// ---- DUTs/IO/PdoEntries/Control_FF5AB9B2.TcDUT
{attribute 'GeneratedUsingTerminal: EJ7334-0008-0016'}
{attribute addProperty BoxType "EJ7334-0008-0016"}
{attribute addProperty Id "EnableBOOL1ResetBOOL1"}
{attribute addProperty CRC "4284135858"}
{attribute addProperty Size "2"}
TYPE Control_FF5AB9B2 :
STRUCT
	{attribute addProperty Name "Enable"}
	Enable : BOOL;
	{attribute addProperty Name "Reset"}
	Reset : BOOL;
END_STRUCT
END_TYPE

// ---- DUTs/IO/PdoEntries/FSOE_1F44E1B4.TcDUT
{attribute 'GeneratedUsingTerminal: EJ1914-0000-0017'}
{attribute addProperty BoxType "EJ1914-0000-0017"}
{attribute addProperty Id "FSoE_CommandUSINT1FSIN_Module_1_Channel_1_InputBOOL1FSIN_Module_1_Channel_2_InputBOOL1FSIN_Module_1_Module_FaultBOOL1FSIN_Module_2_Channel_1_InputBOOL1FSIN_Module_2_Channel_2_InputBOOL1FSIN_Module_2_Module_FaultBOOL1FSoE_CRC_000UINT2FSoE_Connection_IDUINT2"}
{attribute addProperty CRC "524607924"}
{attribute addProperty Size "11"}
TYPE FSOE_1F44E1B4 :
STRUCT
	{attribute addProperty Name "FSoE_Command"}
	FSoE_Command : USINT;
	{attribute addProperty Name "FSIN_Module_1_Channel_1_Input"}
	FSIN_Module_1_Channel_1_Input : BOOL;
	{attribute addProperty Name "FSIN_Module_1_Channel_2_Input"}
	FSIN_Module_1_Channel_2_Input : BOOL;
	{attribute addProperty Name "FSIN_Module_1_Module_Fault"}
	FSIN_Module_1_Module_Fault : BOOL;
	{attribute addProperty Name "FSIN_Module_2_Channel_1_Input"}
	FSIN_Module_2_Channel_1_Input : BOOL;
	{attribute addProperty Name "FSIN_Module_2_Channel_2_Input"}
	FSIN_Module_2_Channel_2_Input : BOOL;
	{attribute addProperty Name "FSIN_Module_2_Module_Fault"}
	FSIN_Module_2_Module_Fault : BOOL;
	{attribute addProperty Name "FSoE_CRC_000"}
	FSoE_CRC_000 : UINT;
	{attribute addProperty Name "FSoE_Connection_ID"}
	FSoE_Connection_ID : UINT;
END_STRUCT
END_TYPE

// ---- DUTs/IO/PdoEntries/FSOE_9A7ED3DD.TcDUT
{attribute 'GeneratedUsingTerminal: EJ1914-0000-0017'}
{attribute addProperty BoxType "EJ1914-0000-0017"}
{attribute addProperty Id "FSoE_CommandUSINT1FSIN_Module_1_ErrAckBOOL1FSIN_Module_2_ErrAckBOOL1FSoE_CRC_000UINT2FSoE_Connection_IDUINT2"}
{attribute addProperty CRC "2592003037"}
{attribute addProperty Size "7"}
TYPE FSOE_9A7ED3DD :
STRUCT
	{attribute addProperty Name "FSoE_Command"}
	FSoE_Command : USINT;
	{attribute addProperty Name "FSIN_Module_1_ErrAck"}
	FSIN_Module_1_ErrAck : BOOL;
	{attribute addProperty Name "FSIN_Module_2_ErrAck"}
	FSIN_Module_2_ErrAck : BOOL;
	{attribute addProperty Name "FSoE_CRC_000"}
	FSoE_CRC_000 : UINT;
	{attribute addProperty Name "FSoE_Connection_ID"}
	FSoE_Connection_ID : UINT;
END_STRUCT
END_TYPE

// ---- DUTs/IO/PdoEntries/FSOE_9F04885D.TcDUT
{attribute 'GeneratedUsingTerminal: EJ1918-0000-0017'}
{attribute addProperty BoxType "EJ1918-0000-0017"}
{attribute addProperty Id "FSoE_CommandUSINT1FSIN_Module_1_Channel_1_InputBOOL1FSIN_Module_1_Channel_2_InputBOOL1FSIN_Module_1_Module_FaultBOOL1FSIN_Module_2_Channel_1_InputBOOL1FSIN_Module_2_Channel_2_InputBOOL1FSIN_Module_2_Module_FaultBOOL1FSIN_Module_3_Channel_1_InputBOOL1FSIN_Module_3_Channel_2_InputBOOL1FSIN_Module_3_Module_FaultBOOL1FSIN_Module_4_Channel_1_InputBOOL1FSIN_Module_4_Channel_2_InputBOOL1FSIN_Module_4_Module_FaultBOOL1FSoE_CRC_000UINT2FSoE_Connection_IDUINT2"}
{attribute addProperty CRC "2667874397"}
{attribute addProperty Size "17"}
TYPE FSOE_9F04885D :
STRUCT
	{attribute addProperty Name "FSoE_Command"}
	FSoE_Command : USINT;
	{attribute addProperty Name "FSIN_Module_1_Channel_1_Input"}
	FSIN_Module_1_Channel_1_Input : BOOL;
	{attribute addProperty Name "FSIN_Module_1_Channel_2_Input"}
	FSIN_Module_1_Channel_2_Input : BOOL;
	{attribute addProperty Name "FSIN_Module_1_Module_Fault"}
	FSIN_Module_1_Module_Fault : BOOL;
	{attribute addProperty Name "FSIN_Module_2_Channel_1_Input"}
	FSIN_Module_2_Channel_1_Input : BOOL;
	{attribute addProperty Name "FSIN_Module_2_Channel_2_Input"}
	FSIN_Module_2_Channel_2_Input : BOOL;
	{attribute addProperty Name "FSIN_Module_2_Module_Fault"}
	FSIN_Module_2_Module_Fault : BOOL;
	{attribute addProperty Name "FSIN_Module_3_Channel_1_Input"}
	FSIN_Module_3_Channel_1_Input : BOOL;
	{attribute addProperty Name "FSIN_Module_3_Channel_2_Input"}
	FSIN_Module_3_Channel_2_Input : BOOL;
	{attribute addProperty Name "FSIN_Module_3_Module_Fault"}
	FSIN_Module_3_Module_Fault : BOOL;
	{attribute addProperty Name "FSIN_Module_4_Channel_1_Input"}
	FSIN_Module_4_Channel_1_Input : BOOL;
	{attribute addProperty Name "FSIN_Module_4_Channel_2_Input"}
	FSIN_Module_4_Channel_2_Input : BOOL;
	{attribute addProperty Name "FSIN_Module_4_Module_Fault"}
	FSIN_Module_4_Module_Fault : BOOL;
	{attribute addProperty Name "FSoE_CRC_000"}
	FSoE_CRC_000 : UINT;
	{attribute addProperty Name "FSoE_Connection_ID"}
	FSoE_Connection_ID : UINT;
END_STRUCT
END_TYPE

// ---- DUTs/IO/PdoEntries/FSOE_87848461.TcDUT
{attribute 'GeneratedUsingTerminal: EJ1918-0000-0017'}
{attribute addProperty BoxType "EJ1918-0000-0017"}
{attribute addProperty Id "FSoE_CommandUSINT1FSIN_Module_1_ErrAckBOOL1FSIN_Module_2_ErrAckBOOL1FSIN_Module_3_ErrAckBOOL1FSIN_Module_4_ErrAckBOOL1FSoE_CRC_000UINT2FSoE_Connection_IDUINT2"}
{attribute addProperty CRC "2273608801"}
{attribute addProperty Size "9"}
TYPE FSOE_87848461 :
STRUCT
	{attribute addProperty Name "FSoE_Command"}
	FSoE_Command : USINT;
	{attribute addProperty Name "FSIN_Module_1_ErrAck"}
	FSIN_Module_1_ErrAck : BOOL;
	{attribute addProperty Name "FSIN_Module_2_ErrAck"}
	FSIN_Module_2_ErrAck : BOOL;
	{attribute addProperty Name "FSIN_Module_3_ErrAck"}
	FSIN_Module_3_ErrAck : BOOL;
	{attribute addProperty Name "FSIN_Module_4_ErrAck"}
	FSIN_Module_4_ErrAck : BOOL;
	{attribute addProperty Name "FSoE_CRC_000"}
	FSoE_CRC_000 : UINT;
	{attribute addProperty Name "FSoE_Connection_ID"}
	FSoE_Connection_ID : UINT;
END_STRUCT
END_TYPE

// ---- DUTs/IO/PdoEntries/FSOE_BBC930F7.TcDUT
{attribute 'GeneratedUsingTerminal: EJ1957-0000-0017'}
{attribute addProperty BoxType "EJ1957-0000-0017"}
{attribute addProperty Id "FSoE_CommandUSINT1FSOUT_Module_Module_FaultBOOL1FSIN_Module_1_Channel_1_InputBOOL1FSIN_Module_1_Channel_2_InputBOOL1FSIN_Module_1_Module_FaultBOOL1FSIN_Module_2_Channel_1_InputBOOL1FSIN_Module_2_Channel_2_InputBOOL1FSIN_Module_2_Module_FaultBOOL1FSIN_Module_3_Channel_1_InputBOOL1FSIN_Module_3_Channel_2_InputBOOL1FSIN_Module_3_Module_FaultBOOL1FSIN_Module_4_Channel_1_InputBOOL1FSIN_Module_4_Channel_2_InputBOOL1FSIN_Module_4_Module_FaultBOOL1FSoE_CRC_000UINT2FSoE_Connection_IDUINT2"}
{attribute addProperty CRC "3150524663"}
{attribute addProperty Size "18"}
TYPE FSOE_BBC930F7 :
STRUCT
	{attribute addProperty Name "FSoE_Command"}
	FSoE_Command : USINT;
	{attribute addProperty Name "FSOUT_Module_Module_Fault"}
	FSOUT_Module_Module_Fault : BOOL;
	{attribute addProperty Name "FSIN_Module_1_Channel_1_Input"}
	FSIN_Module_1_Channel_1_Input : BOOL;
	{attribute addProperty Name "FSIN_Module_1_Channel_2_Input"}
	FSIN_Module_1_Channel_2_Input : BOOL;
	{attribute addProperty Name "FSIN_Module_1_Module_Fault"}
	FSIN_Module_1_Module_Fault : BOOL;
	{attribute addProperty Name "FSIN_Module_2_Channel_1_Input"}
	FSIN_Module_2_Channel_1_Input : BOOL;
	{attribute addProperty Name "FSIN_Module_2_Channel_2_Input"}
	FSIN_Module_2_Channel_2_Input : BOOL;
	{attribute addProperty Name "FSIN_Module_2_Module_Fault"}
	FSIN_Module_2_Module_Fault : BOOL;
	{attribute addProperty Name "FSIN_Module_3_Channel_1_Input"}
	FSIN_Module_3_Channel_1_Input : BOOL;
	{attribute addProperty Name "FSIN_Module_3_Channel_2_Input"}
	FSIN_Module_3_Channel_2_Input : BOOL;
	{attribute addProperty Name "FSIN_Module_3_Module_Fault"}
	FSIN_Module_3_Module_Fault : BOOL;
	{attribute addProperty Name "FSIN_Module_4_Channel_1_Input"}
	FSIN_Module_4_Channel_1_Input : BOOL;
	{attribute addProperty Name "FSIN_Module_4_Channel_2_Input"}
	FSIN_Module_4_Channel_2_Input : BOOL;
	{attribute addProperty Name "FSIN_Module_4_Module_Fault"}
	FSIN_Module_4_Module_Fault : BOOL;
	{attribute addProperty Name "FSoE_CRC_000"}
	FSoE_CRC_000 : UINT;
	{attribute addProperty Name "FSoE_Connection_ID"}
	FSoE_Connection_ID : UINT;
END_STRUCT
END_TYPE

// ---- DUTs/IO/PdoEntries/FSOE_D1C9D1EA.TcDUT
{attribute 'GeneratedUsingTerminal: EJ1957-0000-0017'}
{attribute addProperty BoxType "EJ1957-0000-0017"}
{attribute addProperty Id "FSoE_CommandUSINT1FSOUT_Module_Channel_1_OutputBOOL1FSOUT_Module_Channel_2_OutputBOOL1FSOUT_Module_Channel_3_OutputBOOL1FSOUT_Module_Channel_4_OutputBOOL1FSOUT_Module_ErrAckBOOL1FSIN_Module_1_ErrAckBOOL1FSIN_Module_2_ErrAckBOOL1FSIN_Module_3_ErrAckBOOL1FSIN_Module_4_ErrAckBOOL1FSoE_CRC_000UINT2FSoE_Connection_IDUINT2"}
{attribute addProperty CRC "3519664618"}
{attribute addProperty Size "14"}
TYPE FSOE_D1C9D1EA :
STRUCT
	{attribute addProperty Name "FSoE_Command"}
	FSoE_Command : USINT;
	{attribute addProperty Name "FSOUT_Module_Channel_1_Output"}
	FSOUT_Module_Channel_1_Output : BOOL;
	{attribute addProperty Name "FSOUT_Module_Channel_2_Output"}
	FSOUT_Module_Channel_2_Output : BOOL;
	{attribute addProperty Name "FSOUT_Module_Channel_3_Output"}
	FSOUT_Module_Channel_3_Output : BOOL;
	{attribute addProperty Name "FSOUT_Module_Channel_4_Output"}
	FSOUT_Module_Channel_4_Output : BOOL;
	{attribute addProperty Name "FSOUT_Module_ErrAck"}
	FSOUT_Module_ErrAck : BOOL;
	{attribute addProperty Name "FSIN_Module_1_ErrAck"}
	FSIN_Module_1_ErrAck : BOOL;
	{attribute addProperty Name "FSIN_Module_2_ErrAck"}
	FSIN_Module_2_ErrAck : BOOL;
	{attribute addProperty Name "FSIN_Module_3_ErrAck"}
	FSIN_Module_3_ErrAck : BOOL;
	{attribute addProperty Name "FSIN_Module_4_ErrAck"}
	FSIN_Module_4_ErrAck : BOOL;
	{attribute addProperty Name "FSoE_CRC_000"}
	FSoE_CRC_000 : UINT;
	{attribute addProperty Name "FSoE_Connection_ID"}
	FSoE_Connection_ID : UINT;
END_STRUCT
END_TYPE

// ---- DUTs/IO/PdoEntries/FSOE_D94E700C.TcDUT
{attribute 'GeneratedUsingTerminal: EJ2914-0000-0017'}
{attribute addProperty BoxType "EJ2914-0000-0017"}
{attribute addProperty Id "FSoE_CommandUSINT1FSOUT_Module_Module_FaultBOOL1FSoE_CRC_000UINT2FSoE_Connection_IDUINT2"}
{attribute addProperty CRC "3645796364"}
{attribute addProperty Size "6"}
TYPE FSOE_D94E700C :
STRUCT
	{attribute addProperty Name "FSoE_Command"}
	FSoE_Command : USINT;
	{attribute addProperty Name "FSOUT_Module_Module_Fault"}
	FSOUT_Module_Module_Fault : BOOL;
	{attribute addProperty Name "FSoE_CRC_000"}
	FSoE_CRC_000 : UINT;
	{attribute addProperty Name "FSoE_Connection_ID"}
	FSoE_Connection_ID : UINT;
END_STRUCT
END_TYPE

// ---- DUTs/IO/PdoEntries/FSOE_1DB604F4.TcDUT
{attribute 'GeneratedUsingTerminal: EJ2914-0000-0017'}
{attribute addProperty BoxType "EJ2914-0000-0017"}
{attribute addProperty Id "FSoE_CommandUSINT1FSOUT_Module_Channel_1_OutputBOOL1FSOUT_Module_Channel_2_OutputBOOL1FSOUT_Module_Channel_3_OutputBOOL1FSOUT_Module_Channel_4_OutputBOOL1FSOUT_Module_ErrAckBOOL1FSoE_CRC_000UINT2FSoE_Connection_IDUINT2"}
{attribute addProperty CRC "498468084"}
{attribute addProperty Size "10"}
TYPE FSOE_1DB604F4 :
STRUCT
	{attribute addProperty Name "FSoE_Command"}
	FSoE_Command : USINT;
	{attribute addProperty Name "FSOUT_Module_Channel_1_Output"}
	FSOUT_Module_Channel_1_Output : BOOL;
	{attribute addProperty Name "FSOUT_Module_Channel_2_Output"}
	FSOUT_Module_Channel_2_Output : BOOL;
	{attribute addProperty Name "FSOUT_Module_Channel_3_Output"}
	FSOUT_Module_Channel_3_Output : BOOL;
	{attribute addProperty Name "FSOUT_Module_Channel_4_Output"}
	FSOUT_Module_Channel_4_Output : BOOL;
	{attribute addProperty Name "FSOUT_Module_ErrAck"}
	FSOUT_Module_ErrAck : BOOL;
	{attribute addProperty Name "FSoE_CRC_000"}
	FSoE_CRC_000 : UINT;
	{attribute addProperty Name "FSoE_Connection_ID"}
	FSoE_Connection_ID : UINT;
END_STRUCT
END_TYPE

// ---- DUTs/IO/PdoEntries/FSOE_046F804E.TcDUT
{attribute 'GeneratedUsingTerminal: EJ2918-0000-0017'}
{attribute addProperty BoxType "EJ2918-0000-0017"}
{attribute addProperty Id "FSoE_CommandUSINT1FSOUT_Module_1_Module_FaultBOOL1FSOUT_Module_2_Module_FaultBOOL1FSoE_CRC_000UINT2FSoE_Connection_IDUINT2"}
{attribute addProperty CRC "74416206"}
{attribute addProperty Size "7"}
TYPE FSOE_046F804E :
STRUCT
	{attribute addProperty Name "FSoE_Command"}
	FSoE_Command : USINT;
	{attribute addProperty Name "FSOUT_Module_1_Module_Fault"}
	FSOUT_Module_1_Module_Fault : BOOL;
	{attribute addProperty Name "FSOUT_Module_2_Module_Fault"}
	FSOUT_Module_2_Module_Fault : BOOL;
	{attribute addProperty Name "FSoE_CRC_000"}
	FSoE_CRC_000 : UINT;
	{attribute addProperty Name "FSoE_Connection_ID"}
	FSoE_Connection_ID : UINT;
END_STRUCT
END_TYPE

// ---- DUTs/IO/PdoEntries/FSOE_2DC96D31.TcDUT
{attribute 'GeneratedUsingTerminal: EJ2918-0000-0017'}
{attribute addProperty BoxType "EJ2918-0000-0017"}
{attribute addProperty Id "FSoE_CommandUSINT1FSOUT_Module_1_Channel_1_OutputBOOL1FSOUT_Module_1_Channel_2_OutputBOOL1FSOUT_Module_1_Channel_3_OutputBOOL1FSOUT_Module_1_Channel_4_OutputBOOL1FSOUT_Module_1_ErrAckBOOL1FSOUT_Module_2_Channel_1_OutputBOOL1FSOUT_Module_2_Channel_2_OutputBOOL1FSOUT_Module_2_Channel_3_OutputBOOL1FSOUT_Module_2_Channel_4_OutputBOOL1FSOUT_Module_2_ErrAckBOOL1FSoE_CRC_000UINT2FSoE_Connection_IDUINT2"}
{attribute addProperty CRC "768175409"}
{attribute addProperty Size "15"}
TYPE FSOE_2DC96D31 :
STRUCT
	{attribute addProperty Name "FSoE_Command"}
	FSoE_Command : USINT;
	{attribute addProperty Name "FSOUT_Module_1_Channel_1_Output"}
	FSOUT_Module_1_Channel_1_Output : BOOL;
	{attribute addProperty Name "FSOUT_Module_1_Channel_2_Output"}
	FSOUT_Module_1_Channel_2_Output : BOOL;
	{attribute addProperty Name "FSOUT_Module_1_Channel_3_Output"}
	FSOUT_Module_1_Channel_3_Output : BOOL;
	{attribute addProperty Name "FSOUT_Module_1_Channel_4_Output"}
	FSOUT_Module_1_Channel_4_Output : BOOL;
	{attribute addProperty Name "FSOUT_Module_1_ErrAck"}
	FSOUT_Module_1_ErrAck : BOOL;
	{attribute addProperty Name "FSOUT_Module_2_Channel_1_Output"}
	FSOUT_Module_2_Channel_1_Output : BOOL;
	{attribute addProperty Name "FSOUT_Module_2_Channel_2_Output"}
	FSOUT_Module_2_Channel_2_Output : BOOL;
	{attribute addProperty Name "FSOUT_Module_2_Channel_3_Output"}
	FSOUT_Module_2_Channel_3_Output : BOOL;
	{attribute addProperty Name "FSOUT_Module_2_Channel_4_Output"}
	FSOUT_Module_2_Channel_4_Output : BOOL;
	{attribute addProperty Name "FSOUT_Module_2_ErrAck"}
	FSOUT_Module_2_ErrAck : BOOL;
	{attribute addProperty Name "FSoE_CRC_000"}
	FSoE_CRC_000 : UINT;
	{attribute addProperty Name "FSoE_Connection_ID"}
	FSoE_Connection_ID : UINT;
END_STRUCT
END_TYPE

// ---- DUTs/IO/PDOs/InfoData_6F19DB2B.TcDUT
{attribute 'GeneratedUsingTerminal: EK1100-0000-0018'}
{attribute addProperty BoxType "EK1100-0000-0018"}
{attribute addProperty Id "StateAT %I*UINT2"}
{attribute addProperty CRC "1863965483"}
{attribute addProperty Size "2"}
TYPE InfoData_6F19DB2B :
STRUCT
	{attribute addProperty Name "State"}
	State AT %I* : UINT;
END_STRUCT
END_TYPE

// ---- DUTs/IO/PDOs/WcState_0B2B16F9.TcDUT
{attribute 'GeneratedUsingTerminal: EJ1101-0022-0016'}
{attribute addProperty BoxType "EJ1101-0022-0016"}
{attribute addProperty Id "WcStateAT %I*BOOL1"}
{attribute addProperty CRC "187373305"}
{attribute addProperty Size "1"}
TYPE WcState_0B2B16F9 :
STRUCT
	{attribute addProperty Name "WcState"}
	WcState AT %I* : BOOL;
END_STRUCT
END_TYPE

// ---- DUTs/IO/PDOs/InfoData_32EB74EA.TcDUT
{attribute 'GeneratedUsingTerminal: EJ1101-0022-0016'}
{attribute addProperty BoxType "EJ1101-0022-0016"}
{attribute addProperty Id "AdsAddrAT %I*AMSADDR8StateAT %I*UINT2"}
{attribute addProperty CRC "854291690"}
{attribute addProperty Size "10"}
TYPE InfoData_32EB74EA EXTENDS InputBase_8311D824 :
STRUCT
	{attribute addProperty Name "AdsAddr"}
	AdsAddr AT %I* : AMSADDR;
	{attribute addProperty Name "State"}
	State AT %I* : UINT;
END_STRUCT
END_TYPE

// ---- DUTs/IO/PDOs/Channel_830843C1.TcDUT
{attribute 'GeneratedUsingTerminal: EJ1008-0000-0017'}
{attribute addProperty BoxType "EJ1008-0000-0017"}
{attribute addProperty Id "InputAT %I*BOOL1"}
{attribute addProperty CRC "2198356929"}
{attribute addProperty Size "1"}
TYPE Channel_830843C1 EXTENDS InputBase_8311D824 :
STRUCT
	{attribute addProperty Name "Input"}
	Input AT %I* : BOOL;
END_STRUCT
END_TYPE

// ---- DUTs/IO/PDOs/WcState_9091E0EB.TcDUT
{attribute 'GeneratedUsingTerminal: EJ1008-0000-0017'}
{attribute addProperty BoxType "EJ1008-0000-0017"}
{attribute addProperty Id "WcStateAT %I*BOOL1InputToggleAT %I*BOOL1"}
{attribute addProperty CRC "2425479403"}
{attribute addProperty Size "2"}
TYPE WcState_9091E0EB :
STRUCT
	{attribute addProperty Name "WcState"}
	WcState AT %I* : BOOL;
	{attribute addProperty Name "InputToggle"}
	InputToggle AT %I* : BOOL;
END_STRUCT
END_TYPE

// ---- DUTs/IO/PDOs/Channel_42CA91F7.TcDUT
{attribute 'GeneratedUsingTerminal: EJ1859-0000-0017'}
{attribute addProperty BoxType "EJ1859-0000-0017"}
{attribute addProperty Id "OutputAT %Q*BOOL1"}
{attribute addProperty CRC "1120571895"}
{attribute addProperty Size "1"}
TYPE Channel_42CA91F7 EXTENDS OutputBase_10CEE7DE :
STRUCT
	{attribute addProperty Name "Output"}
	Output AT %Q* : BOOL;
END_STRUCT
END_TYPE

// ---- DUTs/IO/PDOs/PWM_Outputs_Channel_4C6289CD.TcDUT
{attribute 'GeneratedUsingTerminal: EJ2502-0000-0023'}
{attribute addProperty BoxType "EJ2502-0000-0023"}
{attribute addProperty Id "PWM_outputAT %Q*UINT2"}
{attribute addProperty CRC "1281526221"}
{attribute addProperty Size "2"}
TYPE PWM_Outputs_Channel_4C6289CD EXTENDS OutputBase_10CEE7DE :
STRUCT
	{attribute addProperty Name "PWM_output"}
	PWM_output AT %Q* : UINT;
END_STRUCT
END_TYPE

// ---- DUTs/IO/PDOs/PTO_Status_E0EB10E8.TcDUT
{attribute 'GeneratedUsingTerminal: EJ2521-0224-0016'}
{attribute addProperty BoxType "EJ2521-0224-0016"}
{attribute addProperty Id "StatusAT %I*Status_B83811715"}
{attribute addProperty CRC "3773501672"}
{attribute addProperty Size "5"}
TYPE PTO_Status_E0EB10E8 EXTENDS InputBase_8311D824 :
STRUCT
	{attribute addProperty Name "Status"}
	Status AT %I* : Status_B8381171;
END_STRUCT
END_TYPE

// ---- DUTs/IO/PDOs/ENC_Status_compact_3C6E2C44.TcDUT
{attribute 'GeneratedUsingTerminal: EJ2521-0224-0016'}
{attribute addProperty BoxType "EJ2521-0224-0016"}
{attribute addProperty Id "StatusAT %I*Status_182674C67Counter_valueAT %I*UINT2Latch_valueAT %I*UINT2"}
{attribute addProperty CRC "1013853252"}
{attribute addProperty Size "11"}
TYPE ENC_Status_compact_3C6E2C44 EXTENDS InputBase_8311D824 :
STRUCT
	{attribute addProperty Name "Status"}
	Status AT %I* : Status_182674C6;
	{attribute addProperty Name "Counter_value"}
	Counter_value AT %I* : UINT;
	{attribute addProperty Name "Latch_value"}
	Latch_value AT %I* : UINT;
END_STRUCT
END_TYPE

// ---- DUTs/IO/PDOs/PLS_Status_Channel_70E7A1E2.TcDUT
{attribute 'GeneratedUsingTerminal: EJ2521-0224-0016'}
{attribute addProperty BoxType "EJ2521-0224-0016"}
{attribute addProperty Id "StatusAT %I*Status_7097155E4"}
{attribute addProperty CRC "1894228450"}
{attribute addProperty Size "4"}
TYPE PLS_Status_Channel_70E7A1E2 EXTENDS InputBase_8311D824 :
STRUCT
	{attribute addProperty Name "Status"}
	Status AT %I* : Status_7097155E;
END_STRUCT
END_TYPE

// ---- DUTs/IO/PDOs/PTO_Control_9287F8E4.TcDUT
{attribute 'GeneratedUsingTerminal: EJ2521-0224-0016'}
{attribute addProperty BoxType "EJ2521-0224-0016"}
{attribute addProperty Id "ControlAT %Q*Control_DAEE1D523Frequency_valueAT %Q*UINT2"}
{attribute addProperty CRC "2458384612"}
{attribute addProperty Size "5"}
TYPE PTO_Control_9287F8E4 EXTENDS OutputBase_10CEE7DE :
STRUCT
	{attribute addProperty Name "Control"}
	Control AT %Q* : Control_DAEE1D52;
	{attribute addProperty Name "Frequency_value"}
	Frequency_value AT %Q* : UINT;
END_STRUCT
END_TYPE

// ---- DUTs/IO/PDOs/PTO_Target_compact_5C359F7D.TcDUT
{attribute 'GeneratedUsingTerminal: EJ2521-0224-0016'}
{attribute addProperty BoxType "EJ2521-0224-0016"}
{attribute addProperty Id "Target_counter_valueAT %Q*UINT2"}
{attribute addProperty CRC "1547018109"}
{attribute addProperty Size "2"}
TYPE PTO_Target_compact_5C359F7D EXTENDS OutputBase_10CEE7DE :
STRUCT
	{attribute addProperty Name "Target_counter_value"}
	Target_counter_value AT %Q* : UINT;
END_STRUCT
END_TYPE

// ---- DUTs/IO/PDOs/ENC_Control_compact_2E82BC43.TcDUT
{attribute 'GeneratedUsingTerminal: EJ2521-0224-0016'}
{attribute addProperty BoxType "EJ2521-0224-0016"}
{attribute addProperty Id "ControlAT %Q*Control_F189B7373Set_counter_valueAT %Q*UINT2"}
{attribute addProperty CRC "780319811"}
{attribute addProperty Size "5"}
TYPE ENC_Control_compact_2E82BC43 EXTENDS OutputBase_10CEE7DE :
STRUCT
	{attribute addProperty Name "Control"}
	Control AT %Q* : Control_F189B737;
	{attribute addProperty Name "Set_counter_value"}
	Set_counter_value AT %Q* : UINT;
END_STRUCT
END_TYPE

// ---- DUTs/IO/PDOs/PLS_Control_compact_Channel_CD6E44DE.TcDUT
{attribute 'GeneratedUsingTerminal: EJ2521-0224-0016'}
{attribute addProperty BoxType "EJ2521-0224-0016"}
{attribute addProperty Id "ControlAT %Q*Control_7786EF9F2Switch_on_valueAT %Q*UINT2Switch_off_valueAT %Q*UINT2"}
{attribute addProperty CRC "3446555870"}
{attribute addProperty Size "6"}
TYPE PLS_Control_compact_Channel_CD6E44DE EXTENDS OutputBase_10CEE7DE :
STRUCT
	{attribute addProperty Name "Control"}
	Control AT %Q* : Control_7786EF9F;
	{attribute addProperty Name "Switch_on_value"}
	Switch_on_value AT %Q* : UINT;
	{attribute addProperty Name "Switch_off_value"}
	Switch_off_value AT %Q* : UINT;
END_STRUCT
END_TYPE

// ---- DUTs/IO/PDOs/PTO_Status_Channel_E0EB10E8.TcDUT
{attribute 'GeneratedUsingTerminal: EJ2522-0000-0022'}
{attribute addProperty BoxType "EJ2522-0000-0022"}
{attribute addProperty Id "StatusAT %I*Status_B83811715"}
{attribute addProperty CRC "3773501672"}
{attribute addProperty Size "5"}
TYPE PTO_Status_Channel_E0EB10E8 EXTENDS InputBase_8311D824 :
STRUCT
	{attribute addProperty Name "Status"}
	Status AT %I* : Status_B8381171;
END_STRUCT
END_TYPE

// ---- DUTs/IO/PDOs/ENC_Status_Channel_A9252C48.TcDUT
{attribute 'GeneratedUsingTerminal: EJ2522-0000-0022'}
{attribute addProperty BoxType "EJ2522-0000-0022"}
{attribute addProperty Id "StatusAT %I*Status_70E023F86Counter_valueAT %I*UDINT4"}
{attribute addProperty CRC "2837785672"}
{attribute addProperty Size "10"}
TYPE ENC_Status_Channel_A9252C48 EXTENDS InputBase_8311D824 :
STRUCT
	{attribute addProperty Name "Status"}
	Status AT %I* : Status_70E023F8;
	{attribute addProperty Name "Counter_value"}
	Counter_value AT %I* : UDINT;
END_STRUCT
END_TYPE

// ---- DUTs/IO/PDOs/PTO_Control_Channel_9287F8E4.TcDUT
{attribute 'GeneratedUsingTerminal: EJ2522-0000-0022'}
{attribute addProperty BoxType "EJ2522-0000-0022"}
{attribute addProperty Id "ControlAT %Q*Control_DAEE1D523Frequency_valueAT %Q*UINT2"}
{attribute addProperty CRC "2458384612"}
{attribute addProperty Size "5"}
TYPE PTO_Control_Channel_9287F8E4 EXTENDS OutputBase_10CEE7DE :
STRUCT
	{attribute addProperty Name "Control"}
	Control AT %Q* : Control_DAEE1D52;
	{attribute addProperty Name "Frequency_value"}
	Frequency_value AT %Q* : UINT;
END_STRUCT
END_TYPE

// ---- DUTs/IO/PDOs/PTO_Target_Channel_1F6D5BC6.TcDUT
{attribute 'GeneratedUsingTerminal: EJ2522-0000-0022'}
{attribute addProperty BoxType "EJ2522-0000-0022"}
{attribute addProperty Id "Target_counter_valueAT %Q*UDINT4"}
{attribute addProperty CRC "527260614"}
{attribute addProperty Size "4"}
TYPE PTO_Target_Channel_1F6D5BC6 EXTENDS OutputBase_10CEE7DE :
STRUCT
	{attribute addProperty Name "Target_counter_value"}
	Target_counter_value AT %Q* : UDINT;
END_STRUCT
END_TYPE

// ---- DUTs/IO/PDOs/ENC_Control_Channel_686BB9DC.TcDUT
{attribute 'GeneratedUsingTerminal: EJ2522-0000-0022'}
{attribute addProperty BoxType "EJ2522-0000-0022"}
{attribute addProperty Id "ControlAT %Q*Control_A8DDCD822Set_counter_valueAT %Q*UDINT4"}
{attribute addProperty CRC "1751890396"}
{attribute addProperty Size "6"}
TYPE ENC_Control_Channel_686BB9DC EXTENDS OutputBase_10CEE7DE :
STRUCT
	{attribute addProperty Name "Control"}
	Control AT %Q* : Control_A8DDCD82;
	{attribute addProperty Name "Set_counter_value"}
	Set_counter_value AT %Q* : UDINT;
END_STRUCT
END_TYPE

// ---- DUTs/IO/PDOs/AI_Standard_Channel_4A394481.TcDUT
{attribute 'GeneratedUsingTerminal: EJ3004-0000-0019'}
{attribute addProperty BoxType "EJ3004-0000-0019"}
{attribute addProperty Id "StatusAT %I*Status_F2CE6D917ValueAT %I*INT2"}
{attribute addProperty CRC "1245267073"}
{attribute addProperty Size "9"}
TYPE AI_Standard_Channel_4A394481 EXTENDS InputBase_8311D824 :
STRUCT
	{attribute addProperty Name "Status"}
	Status AT %I* : Status_F2CE6D91;
	{attribute addProperty Name "Value"}
	Value AT %I* : INT;
END_STRUCT
END_TYPE

// ---- DUTs/IO/PDOs/AI_Standard_Channel_A8DF64E3.TcDUT
{attribute 'GeneratedUsingTerminal: EJ3104-0000-0019'}
{attribute addProperty BoxType "EJ3104-0000-0019"}
{attribute addProperty Id "StatusAT %I*Status_B07533568ValueAT %I*INT2"}
{attribute addProperty CRC "2833212643"}
{attribute addProperty Size "10"}
TYPE AI_Standard_Channel_A8DF64E3 EXTENDS InputBase_8311D824 :
STRUCT
	{attribute addProperty Name "Status"}
	Status AT %I* : Status_B0753356;
	{attribute addProperty Name "Value"}
	Value AT %I* : INT;
END_STRUCT
END_TYPE

// ---- DUTs/IO/PDOs/RTD_Inputs_Channel_9575FEA1.TcDUT
{attribute 'GeneratedUsingTerminal: EJ3214-0000-0016'}
{attribute addProperty BoxType "EJ3214-0000-0016"}
{attribute addProperty Id "StatusAT %I*Status_68C33E995ValueAT %I*INT2"}
{attribute addProperty CRC "2507538081"}
{attribute addProperty Size "7"}
TYPE RTD_Inputs_Channel_9575FEA1 EXTENDS InputBase_8311D824 :
STRUCT
	{attribute addProperty Name "Status"}
	Status AT %I* : Status_68C33E99;
	{attribute addProperty Name "Value"}
	Value AT %I* : INT;
END_STRUCT
END_TYPE

// ---- DUTs/IO/PDOs/TC_Channel_9575FEA1.TcDUT
{attribute 'GeneratedUsingTerminal: EJ3318-0000-0017'}
{attribute addProperty BoxType "EJ3318-0000-0017"}
{attribute addProperty Id "StatusAT %I*Status_68C33E995ValueAT %I*INT2"}
{attribute addProperty CRC "2507538081"}
{attribute addProperty Size "7"}
TYPE TC_Channel_9575FEA1 EXTENDS InputBase_8311D824 :
STRUCT
	{attribute addProperty Name "Status"}
	Status AT %I* : Status_68C33E99;
	{attribute addProperty Name "Value"}
	Value AT %I* : INT;
END_STRUCT
END_TYPE

// ---- DUTs/IO/PDOs/AO_Output_Channel_BA7EBB7C.TcDUT
{attribute 'GeneratedUsingTerminal: EJ4002-0000-0017'}
{attribute addProperty BoxType "EJ4002-0000-0017"}
{attribute addProperty Id "Analog_outputAT %Q*INT2"}
{attribute addProperty CRC "3128867708"}
{attribute addProperty Size "2"}
TYPE AO_Output_Channel_BA7EBB7C EXTENDS OutputBase_10CEE7DE :
STRUCT
	{attribute addProperty Name "Analog_output"}
	Analog_output AT %Q* : INT;
END_STRUCT
END_TYPE

// ---- DUTs/IO/PDOs/SSI_Inputs_Channel_0E3D8E33.TcDUT
{attribute 'GeneratedUsingTerminal: EJ5002-0000-0016'}
{attribute addProperty BoxType "EJ5002-0000-0016"}
{attribute addProperty Id "StatusAT %I*Status_ACC8459F6Counter_valueAT %I*UDINT4"}
{attribute addProperty CRC "238915123"}
{attribute addProperty Size "10"}
TYPE SSI_Inputs_Channel_0E3D8E33 EXTENDS InputBase_8311D824 :
STRUCT
	{attribute addProperty Name "Status"}
	Status AT %I* : Status_ACC8459F;
	{attribute addProperty Name "Counter_value"}
	Counter_value AT %I* : UDINT;
END_STRUCT
END_TYPE

// ---- DUTs/IO/PDOs/SSI_Inputs_Channel_EDA16284.TcDUT
{attribute 'GeneratedUsingTerminal: EJ5002-0000-0017'}
{attribute addProperty BoxType "EJ5002-0000-0017"}
{attribute addProperty Id "StatusAT %I*Status_C03E24957Counter_valueAT %I*UDINT4"}
{attribute addProperty CRC "3986776708"}
{attribute addProperty Size "11"}
TYPE SSI_Inputs_Channel_EDA16284 EXTENDS InputBase_8311D824 :
STRUCT
	{attribute addProperty Name "Status"}
	Status AT %I* : Status_C03E2495;
	{attribute addProperty Name "Counter_value"}
	Counter_value AT %I* : UDINT;
END_STRUCT
END_TYPE

// ---- DUTs/IO/PDOs/ENC_Status_compact_7D3464F3.TcDUT
{attribute 'GeneratedUsingTerminal: EJ5101-0000-0016'}
{attribute addProperty BoxType "EJ5101-0000-0016"}
{attribute addProperty Id "StatusAT %I*Status_D8D782C316Counter_valueAT %I*UINT2Latch_valueAT %I*UINT2"}
{attribute addProperty CRC "2100585715"}
{attribute addProperty Size "20"}
TYPE ENC_Status_compact_7D3464F3 EXTENDS InputBase_8311D824 :
STRUCT
	{attribute addProperty Name "Status"}
	Status AT %I* : Status_D8D782C3;
	{attribute addProperty Name "Counter_value"}
	Counter_value AT %I* : UINT;
	{attribute addProperty Name "Latch_value"}
	Latch_value AT %I* : UINT;
END_STRUCT
END_TYPE

// ---- DUTs/IO/PDOs/ENC_Control_compact_21E2D14D.TcDUT
{attribute 'GeneratedUsingTerminal: EJ5101-0000-0016'}
{attribute addProperty BoxType "EJ5101-0000-0016"}
{attribute addProperty Id "ControlAT %Q*Control_6EF2C5D04Set_counter_valueAT %Q*UINT2"}
{attribute addProperty CRC "568512845"}
{attribute addProperty Size "6"}
TYPE ENC_Control_compact_21E2D14D EXTENDS OutputBase_10CEE7DE :
STRUCT
	{attribute addProperty Name "Control"}
	Control AT %Q* : Control_6EF2C5D0;
	{attribute addProperty Name "Set_counter_value"}
	Set_counter_value AT %Q* : UINT;
END_STRUCT
END_TYPE

// ---- DUTs/IO/PDOs/ENC_Inputs_B3536485.TcDUT
{attribute 'GeneratedUsingTerminal: EJ5151-0000-0016'}
{attribute addProperty BoxType "EJ5151-0000-0016"}
{attribute addProperty Id "StatusAT %I*Status_3E6F3FF310Counter_valueAT %I*UINT2Latch_valueAT %I*UINT2"}
{attribute addProperty CRC "3008586885"}
{attribute addProperty Size "14"}
TYPE ENC_Inputs_B3536485 EXTENDS InputBase_8311D824 :
STRUCT
	{attribute addProperty Name "Status"}
	Status AT %I* : Status_3E6F3FF3;
	{attribute addProperty Name "Counter_value"}
	Counter_value AT %I* : UINT;
	{attribute addProperty Name "Latch_value"}
	Latch_value AT %I* : UINT;
END_STRUCT
END_TYPE

// ---- DUTs/IO/PDOs/ENC_Inputs_24B63C53.TcDUT
{attribute 'GeneratedUsingTerminal: EJ5151-0000-0016'}
{attribute addProperty BoxType "EJ5151-0000-0016"}
{attribute addProperty Id "Period_valueAT %I*UDINT4"}
{attribute addProperty CRC "615922771"}
{attribute addProperty Size "4"}
TYPE ENC_Inputs_24B63C53 EXTENDS InputBase_8311D824 :
STRUCT
	{attribute addProperty Name "Period_value"}
	Period_value AT %I* : UDINT;
END_STRUCT
END_TYPE

// ---- DUTs/IO/PDOs/ENC_Outputs_21E2D14D.TcDUT
{attribute 'GeneratedUsingTerminal: EJ5151-0000-0016'}
{attribute addProperty BoxType "EJ5151-0000-0016"}
{attribute addProperty Id "ControlAT %Q*Control_6EF2C5D04Set_counter_valueAT %Q*UINT2"}
{attribute addProperty CRC "568512845"}
{attribute addProperty Size "6"}
TYPE ENC_Outputs_21E2D14D EXTENDS OutputBase_10CEE7DE :
STRUCT
	{attribute addProperty Name "Control"}
	Control AT %Q* : Control_6EF2C5D0;
	{attribute addProperty Name "Set_counter_value"}
	Set_counter_value AT %Q* : UINT;
END_STRUCT
END_TYPE

// ---- DUTs/IO/PDOs/COM_Inputs_Channel_3801C95E.TcDUT
{attribute 'GeneratedUsingTerminal: EJ6002-0000-0016'}
{attribute addProperty BoxType "EJ6002-0000-0016"}
{attribute addProperty Id "StatusAT %I*Status_3D84275F8Data_InAT %I*ARRAY[0..21] OF USINT22"}
{attribute addProperty CRC "1334739266"}
{attribute addProperty Size "30"}
TYPE COM_Inputs_Channel_3801C95E EXTENDS InputBase_8311D824 :
STRUCT
	{attribute addProperty Name "Status"}
	Status AT %I* : Status_3D84275F;
	{attribute addProperty Name "Data_In"}
	Data_In AT %I* : ARRAY[0..21] OF USINT;
END_STRUCT
END_TYPE

// ---- DUTs/IO/PDOs/COM_Outputs_Channel_EADA2E0D.TcDUT
{attribute 'GeneratedUsingTerminal: EJ6002-0000-0016'}
{attribute addProperty BoxType "EJ6002-0000-0016"}
{attribute addProperty Id "CtrlAT %Q*Ctrl_1EFB4D3B5Data_OutAT %Q*ARRAY[0..21] OF USINT22"}
{attribute addProperty CRC "3494673196"}
{attribute addProperty Size "27"}
TYPE COM_Outputs_Channel_EADA2E0D EXTENDS OutputBase_10CEE7DE :
STRUCT
	{attribute addProperty Name "Ctrl"}
	Ctrl AT %Q* : Ctrl_1EFB4D3B;
	{attribute addProperty Name "Data_Out"}
	Data_Out AT %Q* : ARRAY[0..21] OF USINT;
END_STRUCT
END_TYPE

// ---- DUTs/IO/PDOs/DeviceState_Inputs_Device_A1210598.TcDUT
{attribute 'GeneratedUsingTerminal: EJ6224-0000-0016'}
{attribute addProperty BoxType "EJ6224-0000-0016"}
{attribute addProperty Id "Device_DiagAT %I*BOOL1Device_StateAT %I*BOOL1"}
{attribute addProperty CRC "2703295896"}
{attribute addProperty Size "2"}
TYPE DeviceState_Inputs_Device_A1210598 EXTENDS InputBase_8311D824 :
STRUCT
	{attribute addProperty Name "Device_Diag"}
	Device_Diag AT %I* : BOOL;
	{attribute addProperty Name "Device_State"}
	Device_State AT %I* : BOOL;
END_STRUCT
END_TYPE

// ---- DUTs/IO/PDOs/DeviceState_Inputs_4751FF76.TcDUT
{attribute 'GeneratedUsingTerminal: EJ6224-0000-0016'}
{attribute addProperty BoxType "EJ6224-0000-0016"}
{attribute addProperty Id "State_Ch1AT %I*USINT1State_Ch2AT %I*USINT1State_Ch3AT %I*USINT1State_Ch4AT %I*USINT1"}
{attribute addProperty CRC "1196556150"}
{attribute addProperty Size "4"}
TYPE DeviceState_Inputs_4751FF76 EXTENDS InputBase_8311D824 :
STRUCT
	{attribute addProperty Name "State_Ch1"}
	State_Ch1 AT %I* : USINT;
	{attribute addProperty Name "State_Ch2"}
	State_Ch2 AT %I* : USINT;
	{attribute addProperty Name "State_Ch3"}
	State_Ch3 AT %I* : USINT;
	{attribute addProperty Name "State_Ch4"}
	State_Ch4 AT %I* : USINT;
END_STRUCT
END_TYPE

// ---- DUTs/IO/PDOs/InfoData_90184F0C.TcDUT
{attribute 'GeneratedUsingTerminal: EJ6224-0000-0016'}
{attribute addProperty BoxType "EJ6224-0000-0016"}
{attribute addProperty Id "AdsAddrAT %I*AMSADDR8AoeNetIdAT %I*AMSNETID6StateAT %I*UINT2"}
{attribute addProperty CRC "2417512204"}
{attribute addProperty Size "16"}
TYPE InfoData_90184F0C EXTENDS InputBase_8311D824 :
STRUCT
	{attribute addProperty Name "AdsAddr"}
	AdsAddr AT %I* : AMSADDR;
	{attribute addProperty Name "AoeNetId"}
	AoeNetId AT %I* : AMSNETID;
	{attribute addProperty Name "State"}
	State AT %I* : UINT;
END_STRUCT
END_TYPE

// ---- DUTs/IO/PDOs/Module_1_DeviceState_Inputs_Device_5322301C.TcDUT
{attribute 'GeneratedUsingTerminal: EJ6224-0000-0016'}
{attribute addProperty BoxType "EJ6224-0000-0016"}
{attribute addProperty Id "DeviceState_Inputs_DeviceDeviceState_Inputs_Device_A12105982"}
{attribute addProperty CRC "1394749468"}
{attribute addProperty Size "2"}
TYPE Module_1_DeviceState_Inputs_Device_5322301C :
STRUCT
	{attribute addProperty Name "DeviceState_Inputs_Device"}
	DeviceState_Inputs_Device  : DeviceState_Inputs_Device_A1210598;
END_STRUCT
END_TYPE

// ---- DUTs/IO/PDOs/Module_2_DeviceState_Inputs_BD6C7035.TcDUT
{attribute 'GeneratedUsingTerminal: EJ6224-0000-0016'}
{attribute addProperty BoxType "EJ6224-0000-0016"}
{attribute addProperty Id "DeviceState_InputsDeviceState_Inputs_4751FF764"}
{attribute addProperty CRC "3178000437"}
{attribute addProperty Size "4"}
TYPE Module_2_DeviceState_Inputs_BD6C7035 :
STRUCT
	{attribute addProperty Name "DeviceState_Inputs"}
	DeviceState_Inputs  : DeviceState_Inputs_4751FF76;
END_STRUCT
END_TYPE

// ---- DUTs/IO/PDOs/STM_Status_36ED096F.TcDUT
{attribute 'GeneratedUsingTerminal: EJ7031-0000-0026'}
{attribute addProperty BoxType "EJ7031-0000-0026"}
{attribute addProperty Id "StatusAT %I*Status_B679584511"}
{attribute addProperty CRC "921504111"}
{attribute addProperty Size "11"}
TYPE STM_Status_36ED096F EXTENDS InputBase_8311D824 :
STRUCT
	{attribute addProperty Name "Status"}
	Status AT %I* : Status_B6795845;
END_STRUCT
END_TYPE

// ---- DUTs/IO/PDOs/STM_Control_5A8B5016.TcDUT
{attribute 'GeneratedUsingTerminal: EJ7031-0000-0026'}
{attribute addProperty BoxType "EJ7031-0000-0026"}
{attribute addProperty Id "ControlAT %Q*Control_C948E0F23"}
{attribute addProperty CRC "1519079446"}
{attribute addProperty Size "3"}
TYPE STM_Control_5A8B5016 EXTENDS OutputBase_10CEE7DE :
STRUCT
	{attribute addProperty Name "Control"}
	Control AT %Q* : Control_C948E0F2;
END_STRUCT
END_TYPE

// ---- DUTs/IO/PDOs/STM_Velocity_A47A3F41.TcDUT
{attribute 'GeneratedUsingTerminal: EJ7031-0000-0026'}
{attribute addProperty BoxType "EJ7031-0000-0026"}
{attribute addProperty Id "VelocityAT %Q*INT2"}
{attribute addProperty CRC "2759475009"}
{attribute addProperty Size "2"}
TYPE STM_Velocity_A47A3F41 EXTENDS OutputBase_10CEE7DE :
STRUCT
	{attribute addProperty Name "Velocity"}
	Velocity AT %Q* : INT;
END_STRUCT
END_TYPE

// ---- DUTs/IO/PDOs/InfoData_6538CF5F.TcDUT
{attribute 'GeneratedUsingTerminal: EJ7031-0000-0026'}
{attribute addProperty BoxType "EJ7031-0000-0026"}
{attribute addProperty Id "AdsAddrAT %I*AMSADDR8Chn0AT %I*USINT1Chn1AT %I*USINT1StateAT %I*UINT2"}
{attribute addProperty CRC "1698221919"}
{attribute addProperty Size "12"}
TYPE InfoData_6538CF5F EXTENDS InputBase_8311D824 :
STRUCT
	{attribute addProperty Name "AdsAddr"}
	AdsAddr AT %I* : AMSADDR;
	{attribute addProperty Name "Chn0"}
	Chn0 AT %I* : USINT;
	{attribute addProperty Name "Chn1"}
	Chn1 AT %I* : USINT;
	{attribute addProperty Name "State"}
	State AT %I* : UINT;
END_STRUCT
END_TYPE

// ---- DUTs/IO/PDOs/ENC_Status_compact_4D066E1A.TcDUT
{attribute 'GeneratedUsingTerminal: EJ7037-0000-0020'}
{attribute addProperty BoxType "EJ7037-0000-0020"}
{attribute addProperty Id "StatusAT %I*Status_8CBE219F12Counter_valueAT %I*UINT2Latch_valueAT %I*UINT2"}
{attribute addProperty CRC "1292267034"}
{attribute addProperty Size "16"}
TYPE ENC_Status_compact_4D066E1A EXTENDS InputBase_8311D824 :
STRUCT
	{attribute addProperty Name "Status"}
	Status AT %I* : Status_8CBE219F;
	{attribute addProperty Name "Counter_value"}
	Counter_value AT %I* : UINT;
	{attribute addProperty Name "Latch_value"}
	Latch_value AT %I* : UINT;
END_STRUCT
END_TYPE

// ---- DUTs/IO/PDOs/STM_Status_DE0D6B37.TcDUT
{attribute 'GeneratedUsingTerminal: EJ7037-0000-0020'}
{attribute addProperty BoxType "EJ7037-0000-0020"}
{attribute addProperty Id "StatusAT %I*Status_1E008DB912"}
{attribute addProperty CRC "3725421367"}
{attribute addProperty Size "12"}
TYPE STM_Status_DE0D6B37 EXTENDS InputBase_8311D824 :
STRUCT
	{attribute addProperty Name "Status"}
	Status AT %I* : Status_1E008DB9;
END_STRUCT
END_TYPE

// ---- DUTs/IO/PDOs/STM_Control_BA4CE352.TcDUT
{attribute 'GeneratedUsingTerminal: EJ7037-0000-0020'}
{attribute addProperty BoxType "EJ7037-0000-0020"}
{attribute addProperty Id "ControlAT %Q*Control_5FD4673D4"}
{attribute addProperty CRC "3125601106"}
{attribute addProperty Size "4"}
TYPE STM_Control_BA4CE352 EXTENDS OutputBase_10CEE7DE :
STRUCT
	{attribute addProperty Name "Control"}
	Control AT %Q* : Control_5FD4673D;
END_STRUCT
END_TYPE

// ---- DUTs/IO/PDOs/ENC_Status_compact_Channel_DC559AB0.TcDUT
{attribute 'GeneratedUsingTerminal: EJ7342-0000-0019'}
{attribute addProperty BoxType "EJ7342-0000-0019"}
{attribute addProperty Id "StatusAT %I*Status_3035BE2E10Counter_valueAT %I*UINT2Latch_valueAT %I*UINT2"}
{attribute addProperty CRC "3696597680"}
{attribute addProperty Size "14"}
TYPE ENC_Status_compact_Channel_DC559AB0 EXTENDS InputBase_8311D824 :
STRUCT
	{attribute addProperty Name "Status"}
	Status AT %I* : Status_3035BE2E;
	{attribute addProperty Name "Counter_value"}
	Counter_value AT %I* : UINT;
	{attribute addProperty Name "Latch_value"}
	Latch_value AT %I* : UINT;
END_STRUCT
END_TYPE

// ---- DUTs/IO/PDOs/DCM_Status_Channel_36ED096F.TcDUT
{attribute 'GeneratedUsingTerminal: EJ7342-0000-0019'}
{attribute addProperty BoxType "EJ7342-0000-0019"}
{attribute addProperty Id "StatusAT %I*Status_B679584511"}
{attribute addProperty CRC "921504111"}
{attribute addProperty Size "11"}
TYPE DCM_Status_Channel_36ED096F EXTENDS InputBase_8311D824 :
STRUCT
	{attribute addProperty Name "Status"}
	Status AT %I* : Status_B6795845;
END_STRUCT
END_TYPE

// ---- DUTs/IO/PDOs/ENC_Control_compact_Channel_2E82BC43.TcDUT
{attribute 'GeneratedUsingTerminal: EJ7342-0000-0019'}
{attribute addProperty BoxType "EJ7342-0000-0019"}
{attribute addProperty Id "ControlAT %Q*Control_F189B7373Set_counter_valueAT %Q*UINT2"}
{attribute addProperty CRC "780319811"}
{attribute addProperty Size "5"}
TYPE ENC_Control_compact_Channel_2E82BC43 EXTENDS OutputBase_10CEE7DE :
STRUCT
	{attribute addProperty Name "Control"}
	Control AT %Q* : Control_F189B737;
	{attribute addProperty Name "Set_counter_value"}
	Set_counter_value AT %Q* : UINT;
END_STRUCT
END_TYPE

// ---- DUTs/IO/PDOs/DCM_Control_Channel_5A8B5016.TcDUT
{attribute 'GeneratedUsingTerminal: EJ7342-0000-0019'}
{attribute addProperty BoxType "EJ7342-0000-0019"}
{attribute addProperty Id "ControlAT %Q*Control_C948E0F23"}
{attribute addProperty CRC "1519079446"}
{attribute addProperty Size "3"}
TYPE DCM_Control_Channel_5A8B5016 EXTENDS OutputBase_10CEE7DE :
STRUCT
	{attribute addProperty Name "Control"}
	Control AT %Q* : Control_C948E0F2;
END_STRUCT
END_TYPE

// ---- DUTs/IO/PDOs/DCM_Velocity_Channel_A47A3F41.TcDUT
{attribute 'GeneratedUsingTerminal: EJ7342-0000-0019'}
{attribute addProperty BoxType "EJ7342-0000-0019"}
{attribute addProperty Id "VelocityAT %Q*INT2"}
{attribute addProperty CRC "2759475009"}
{attribute addProperty Size "2"}
TYPE DCM_Velocity_Channel_A47A3F41 EXTENDS OutputBase_10CEE7DE :
STRUCT
	{attribute addProperty Name "Velocity"}
	Velocity AT %Q* : INT;
END_STRUCT
END_TYPE

// ---- DUTs/IO/PDOs/InfoData_939F71B6.TcDUT
{attribute 'GeneratedUsingTerminal: EJ7342-0000-0019'}
{attribute addProperty BoxType "EJ7342-0000-0019"}
{attribute addProperty Id "AdsAddrAT %I*AMSADDR8Chn0AT %I*USINT1Chn1AT %I*USINT1Chn2AT %I*USINT1Chn3AT %I*USINT1StateAT %I*UINT2"}
{attribute addProperty CRC "2476700086"}
{attribute addProperty Size "14"}
TYPE InfoData_939F71B6 EXTENDS InputBase_8311D824 :
STRUCT
	{attribute addProperty Name "AdsAddr"}
	AdsAddr AT %I* : AMSADDR;
	{attribute addProperty Name "Chn0"}
	Chn0 AT %I* : USINT;
	{attribute addProperty Name "Chn1"}
	Chn1 AT %I* : USINT;
	{attribute addProperty Name "Chn2"}
	Chn2 AT %I* : USINT;
	{attribute addProperty Name "Chn3"}
	Chn3 AT %I* : USINT;
	{attribute addProperty Name "State"}
	State AT %I* : UINT;
END_STRUCT
END_TYPE

// ---- DUTs/IO/PDOs/FB_Position_3FA094ED.TcDUT
{attribute 'GeneratedUsingTerminal: EJ7211-0010-0026'}
{attribute addProperty BoxType "EJ7211-0010-0026"}
{attribute addProperty Id "PositionAT %I*UDINT4"}
{attribute addProperty CRC "1067488493"}
{attribute addProperty Size "4"}
TYPE FB_Position_3FA094ED EXTENDS InputBase_8311D824 :
STRUCT
	{attribute addProperty Name "Position"}
	Position AT %I* : UDINT;
END_STRUCT
END_TYPE

// ---- DUTs/IO/PDOs/DRV_Statusword_9B36FDFC.TcDUT
{attribute 'GeneratedUsingTerminal: EJ7211-0010-0026'}
{attribute addProperty BoxType "EJ7211-0010-0026"}
{attribute addProperty Id "StatuswordAT %I*UINT2"}
{attribute addProperty CRC "2604072444"}
{attribute addProperty Size "2"}
TYPE DRV_Statusword_9B36FDFC EXTENDS InputBase_8311D824 :
STRUCT
	{attribute addProperty Name "Statusword"}
	Statusword AT %I* : UINT;
END_STRUCT
END_TYPE

// ---- DUTs/IO/PDOs/DRV_Controlword_F3F14721.TcDUT
{attribute 'GeneratedUsingTerminal: EJ7211-0010-0026'}
{attribute addProperty BoxType "EJ7211-0010-0026"}
{attribute addProperty Id "ControlwordAT %Q*UINT2"}
{attribute addProperty CRC "4092675873"}
{attribute addProperty Size "2"}
TYPE DRV_Controlword_F3F14721 EXTENDS OutputBase_10CEE7DE :
STRUCT
	{attribute addProperty Name "Controlword"}
	Controlword AT %Q* : UINT;
END_STRUCT
END_TYPE

// ---- DUTs/IO/PDOs/DRV_Target_velocity_08A9583B.TcDUT
{attribute 'GeneratedUsingTerminal: EJ7211-0010-0026'}
{attribute addProperty BoxType "EJ7211-0010-0026"}
{attribute addProperty Id "Target_velocityAT %Q*DINT4"}
{attribute addProperty CRC "145315899"}
{attribute addProperty Size "4"}
TYPE DRV_Target_velocity_08A9583B EXTENDS OutputBase_10CEE7DE :
STRUCT
	{attribute addProperty Name "Target_velocity"}
	Target_velocity AT %Q* : DINT;
END_STRUCT
END_TYPE

// ---- DUTs/IO/PDOs/InfoData_96C94FAE.TcDUT
{attribute 'GeneratedUsingTerminal: EJ7211-0010-0026'}
{attribute addProperty BoxType "EJ7211-0010-0026"}
{attribute addProperty Id "AdsAddrAT %I*AMSADDR8DcOutputShiftAT %I*DINT4DcInputShiftAT %I*DINT4Chn0AT %I*USINT1StateAT %I*UINT2"}
{attribute addProperty CRC "2529775534"}
{attribute addProperty Size "19"}
TYPE InfoData_96C94FAE EXTENDS InputBase_8311D824 :
STRUCT
	{attribute addProperty Name "AdsAddr"}
	AdsAddr AT %I* : AMSADDR;
	{attribute addProperty Name "DcOutputShift"}
	DcOutputShift AT %I* : DINT;
	{attribute addProperty Name "DcInputShift"}
	DcInputShift AT %I* : DINT;
	{attribute addProperty Name "Chn0"}
	Chn0 AT %I* : USINT;
	{attribute addProperty Name "State"}
	State AT %I* : UINT;
END_STRUCT
END_TYPE

// ---- DUTs/IO/PDOs/InfoData_6185D47C.TcDUT
{attribute 'GeneratedUsingTerminal: EJ7211-0010-0030'}
{attribute addProperty BoxType "EJ7211-0010-0030"}
{attribute addProperty Id "AdsAddrAT %I*AMSADDR8DcOutputShiftAT %I*DINT4DcInputShiftAT %I*DINT4Chn0AT %I*USINT1Chn1AT %I*USINT1StateAT %I*UINT2"}
{attribute addProperty CRC "1636160636"}
{attribute addProperty Size "20"}
TYPE InfoData_6185D47C EXTENDS InputBase_8311D824 :
STRUCT
	{attribute addProperty Name "AdsAddr"}
	AdsAddr AT %I* : AMSADDR;
	{attribute addProperty Name "DcOutputShift"}
	DcOutputShift AT %I* : DINT;
	{attribute addProperty Name "DcInputShift"}
	DcInputShift AT %I* : DINT;
	{attribute addProperty Name "Chn0"}
	Chn0 AT %I* : USINT;
	{attribute addProperty Name "Chn1"}
	Chn1 AT %I* : USINT;
	{attribute addProperty Name "State"}
	State AT %I* : UINT;
END_STRUCT
END_TYPE

// ---- DUTs/IO/PDOs/DS402_Statusword_9B36FDFC.TcDUT
{attribute 'GeneratedUsingTerminal: EJ7211-0011-0026'}
{attribute addProperty BoxType "EJ7211-0011-0026"}
{attribute addProperty Id "StatuswordAT %I*UINT2"}
{attribute addProperty CRC "2604072444"}
{attribute addProperty Size "2"}
TYPE DS402_Statusword_9B36FDFC EXTENDS InputBase_8311D824 :
STRUCT
	{attribute addProperty Name "Statusword"}
	Statusword AT %I* : UINT;
END_STRUCT
END_TYPE

// ---- DUTs/IO/PDOs/DS402_Position_actual_value_07DC4C74.TcDUT
{attribute 'GeneratedUsingTerminal: EJ7211-0011-0026'}
{attribute addProperty BoxType "EJ7211-0011-0026"}
{attribute addProperty Id "Position_actual_valueAT %I*UDINT4"}
{attribute addProperty CRC "131878004"}
{attribute addProperty Size "4"}
TYPE DS402_Position_actual_value_07DC4C74 EXTENDS InputBase_8311D824 :
STRUCT
	{attribute addProperty Name "Position_actual_value"}
	Position_actual_value AT %I* : UDINT;
END_STRUCT
END_TYPE

// ---- DUTs/IO/PDOs/DS402_Controlword_F3F14721.TcDUT
{attribute 'GeneratedUsingTerminal: EJ7211-0011-0026'}
{attribute addProperty BoxType "EJ7211-0011-0026"}
{attribute addProperty Id "ControlwordAT %Q*UINT2"}
{attribute addProperty CRC "4092675873"}
{attribute addProperty Size "2"}
TYPE DS402_Controlword_F3F14721 EXTENDS OutputBase_10CEE7DE :
STRUCT
	{attribute addProperty Name "Controlword"}
	Controlword AT %Q* : UINT;
END_STRUCT
END_TYPE

// ---- DUTs/IO/PDOs/DS402_Target_velocity_08A9583B.TcDUT
{attribute 'GeneratedUsingTerminal: EJ7211-0011-0026'}
{attribute addProperty BoxType "EJ7211-0011-0026"}
{attribute addProperty Id "Target_velocityAT %Q*DINT4"}
{attribute addProperty CRC "145315899"}
{attribute addProperty Size "4"}
TYPE DS402_Target_velocity_08A9583B EXTENDS OutputBase_10CEE7DE :
STRUCT
	{attribute addProperty Name "Target_velocity"}
	Target_velocity AT %Q* : DINT;
END_STRUCT
END_TYPE

// ---- DUTs/IO/PDOs/InfoData_8300A75E.TcDUT
{attribute 'GeneratedUsingTerminal: EJ7211-9414-0030'}
{attribute addProperty BoxType "EJ7211-9414-0030"}
{attribute addProperty Id "AdsAddrAT %I*AMSADDR8DcOutputShiftAT %I*DINT4DcInputShiftAT %I*DINT4Chn0AT %I*USINT1Chn1AT %I*USINT1Chn2AT %I*USINT1StateAT %I*UINT2"}
{attribute addProperty CRC "2197858142"}
{attribute addProperty Size "21"}
TYPE InfoData_8300A75E EXTENDS InputBase_8311D824 :
STRUCT
	{attribute addProperty Name "AdsAddr"}
	AdsAddr AT %I* : AMSADDR;
	{attribute addProperty Name "DcOutputShift"}
	DcOutputShift AT %I* : DINT;
	{attribute addProperty Name "DcInputShift"}
	DcInputShift AT %I* : DINT;
	{attribute addProperty Name "Chn0"}
	Chn0 AT %I* : USINT;
	{attribute addProperty Name "Chn1"}
	Chn1 AT %I* : USINT;
	{attribute addProperty Name "Chn2"}
	Chn2 AT %I* : USINT;
	{attribute addProperty Name "State"}
	State AT %I* : UINT;
END_STRUCT
END_TYPE

// ---- DUTs/IO/PDOs/DCM_Status_Channel_45521CDC.TcDUT
{attribute 'GeneratedUsingTerminal: EJ7334-0008-0016'}
{attribute addProperty BoxType "EJ7334-0008-0016"}
{attribute addProperty Id "StatusAT %I*Status_2569232E8"}
{attribute addProperty CRC "1163009244"}
{attribute addProperty Size "8"}
TYPE DCM_Status_Channel_45521CDC EXTENDS InputBase_8311D824 :
STRUCT
	{attribute addProperty Name "Status"}
	Status AT %I* : Status_2569232E;
END_STRUCT
END_TYPE

// ---- DUTs/IO/PDOs/DCM_Outputs_Channel_F77F51CE.TcDUT
{attribute 'GeneratedUsingTerminal: EJ7334-0008-0016'}
{attribute addProperty BoxType "EJ7334-0008-0016"}
{attribute addProperty Id "ControlAT %Q*Control_FF5AB9B22VelocityAT %Q*INT2"}
{attribute addProperty CRC "4152316366"}
{attribute addProperty Size "4"}
TYPE DCM_Outputs_Channel_F77F51CE EXTENDS OutputBase_10CEE7DE :
STRUCT
	{attribute addProperty Name "Control"}
	Control AT %Q* : Control_FF5AB9B2;
	{attribute addProperty Name "Velocity"}
	Velocity AT %Q* : INT;
END_STRUCT
END_TYPE

// ---- DUTs/IO/PDOs/DRV_Following_error_actual_value_5AA320BF.TcDUT
{attribute 'GeneratedUsingTerminal: EJ7411-0000-0018'}
{attribute addProperty BoxType "EJ7411-0000-0018"}
{attribute addProperty Id "Following_error_actual_valueAT %I*DINT4"}
{attribute addProperty CRC "1520640191"}
{attribute addProperty Size "4"}
TYPE DRV_Following_error_actual_value_5AA320BF EXTENDS InputBase_8311D824 :
STRUCT
	{attribute addProperty Name "Following_error_actual_value"}
	Following_error_actual_value AT %I* : DINT;
END_STRUCT
END_TYPE

// ---- DUTs/IO/PDOs/DRV_Target_position_05240F14.TcDUT
{attribute 'GeneratedUsingTerminal: EJ7411-0000-0018'}
{attribute addProperty BoxType "EJ7411-0000-0018"}
{attribute addProperty Id "Target_positionAT %Q*UDINT4"}
{attribute addProperty CRC "86249236"}
{attribute addProperty Size "4"}
TYPE DRV_Target_position_05240F14 EXTENDS OutputBase_10CEE7DE :
STRUCT
	{attribute addProperty Name "Target_position"}
	Target_position AT %Q* : UDINT;
END_STRUCT
END_TYPE

// ---- DUTs/IO/PDOs/Status_Uo_B8D9F2FA.TcDUT
{attribute 'GeneratedUsingTerminal: EJ9505-0000-0016'}
{attribute addProperty BoxType "EJ9505-0000-0016"}
{attribute addProperty Id "Power_OKAT %I*BOOL1OverloadAT %I*BOOL1"}
{attribute addProperty CRC "3101291258"}
{attribute addProperty Size "2"}
TYPE Status_Uo_B8D9F2FA EXTENDS InputBase_8311D824 :
STRUCT
	{attribute addProperty Name "Power_OK"}
	Power_OK AT %I* : BOOL;
	{attribute addProperty Name "Overload"}
	Overload AT %I* : BOOL;
END_STRUCT
END_TYPE

// ---- DUTs/IO/PDOs/BCT_Inputs_8E55234D.TcDUT
{attribute 'GeneratedUsingTerminal: EJ9576-0000-0018'}
{attribute addProperty BoxType "EJ9576-0000-0018"}
{attribute addProperty Id "Terminal_OvertemperatureAT %I*BOOL1I2T_errorAT %I*BOOL1I2T_warningAT %I*BOOL1OvervoltageAT %I*BOOL1UndervoltageAT %I*BOOL1Chopper_onAT %I*BOOL1Input_cycle_counterAT %I*BYTE1DC_link_voltageAT %I*UDINT4Resistor_currentAT %I*DINT4Duty_cylceAT %I*USINT1"}
{attribute addProperty CRC "2387944269"}
{attribute addProperty Size "16"}
TYPE BCT_Inputs_8E55234D EXTENDS InputBase_8311D824 :
STRUCT
	{attribute addProperty Name "Terminal_Overtemperature"}
	Terminal_Overtemperature AT %I* : BOOL;
	{attribute addProperty Name "I2T_error"}
	I2T_error AT %I* : BOOL;
	{attribute addProperty Name "I2T_warning"}
	I2T_warning AT %I* : BOOL;
	{attribute addProperty Name "Overvoltage"}
	Overvoltage AT %I* : BOOL;
	{attribute addProperty Name "Undervoltage"}
	Undervoltage AT %I* : BOOL;
	{attribute addProperty Name "Chopper_on"}
	Chopper_on AT %I* : BOOL;
	{attribute addProperty Name "Input_cycle_counter"}
	Input_cycle_counter AT %I* : BYTE;
	{attribute addProperty Name "DC_link_voltage"}
	DC_link_voltage AT %I* : UDINT;
	{attribute addProperty Name "Resistor_current"}
	Resistor_current AT %I* : DINT;
	{attribute addProperty Name "Duty_cylce"}
	Duty_cylce AT %I* : USINT;
END_STRUCT
END_TYPE

// ---- DUTs/IO/PDOs/BCT_Inputs_4B987895.TcDUT
{attribute 'GeneratedUsingTerminal: EJ9576-0000-0019'}
{attribute addProperty BoxType "EJ9576-0000-0019"}
{attribute addProperty Id "Terminal_OvertemperatureAT %I*BOOL1I2T_errorAT %I*BOOL1I2T_warningAT %I*BOOL1OvervoltageAT %I*BOOL1UndervoltageAT %I*BOOL1Chopper_onAT %I*BOOL1Input_cycle_counterAT %I*BYTE1DC_link_voltageAT %I*UDINT4Resistor_currentAT %I*DINT4Duty_cylceAT %I*USINT1I2T_load_factorAT %I*USINT1"}
{attribute addProperty CRC "1268283541"}
{attribute addProperty Size "17"}
TYPE BCT_Inputs_4B987895 EXTENDS InputBase_8311D824 :
STRUCT
	{attribute addProperty Name "Terminal_Overtemperature"}
	Terminal_Overtemperature AT %I* : BOOL;
	{attribute addProperty Name "I2T_error"}
	I2T_error AT %I* : BOOL;
	{attribute addProperty Name "I2T_warning"}
	I2T_warning AT %I* : BOOL;
	{attribute addProperty Name "Overvoltage"}
	Overvoltage AT %I* : BOOL;
	{attribute addProperty Name "Undervoltage"}
	Undervoltage AT %I* : BOOL;
	{attribute addProperty Name "Chopper_on"}
	Chopper_on AT %I* : BOOL;
	{attribute addProperty Name "Input_cycle_counter"}
	Input_cycle_counter AT %I* : BYTE;
	{attribute addProperty Name "DC_link_voltage"}
	DC_link_voltage AT %I* : UDINT;
	{attribute addProperty Name "Resistor_current"}
	Resistor_current AT %I* : DINT;
	{attribute addProperty Name "Duty_cylce"}
	Duty_cylce AT %I* : USINT;
	{attribute addProperty Name "I2T_load_factor"}
	I2T_load_factor AT %I* : USINT;
END_STRUCT
END_TYPE

// ---- DUTs/IO/PDOs/BCT_Inputs_8B1D510C.TcDUT
{attribute 'GeneratedUsingTerminal: EJ9576-0000-0020'}
{attribute addProperty BoxType "EJ9576-0000-0020"}
{attribute addProperty Id "Terminal_OvertemperatureAT %I*BOOL1I2T_errorAT %I*BOOL1I2T_warningAT %I*BOOL1OvervoltageAT %I*BOOL1UndervoltageAT %I*BOOL1Chopper_onAT %I*BOOL1Input_cycle_counterAT %I*BYTE1DC_link_voltageAT %I*UDINT4Resistor_CurrentAT %I*DINT4Duty_CycleAT %I*USINT1"}
{attribute addProperty CRC "2333954316"}
{attribute addProperty Size "16"}
TYPE BCT_Inputs_8B1D510C EXTENDS InputBase_8311D824 :
STRUCT
	{attribute addProperty Name "Terminal_Overtemperature"}
	Terminal_Overtemperature AT %I* : BOOL;
	{attribute addProperty Name "I2T_error"}
	I2T_error AT %I* : BOOL;
	{attribute addProperty Name "I2T_warning"}
	I2T_warning AT %I* : BOOL;
	{attribute addProperty Name "Overvoltage"}
	Overvoltage AT %I* : BOOL;
	{attribute addProperty Name "Undervoltage"}
	Undervoltage AT %I* : BOOL;
	{attribute addProperty Name "Chopper_on"}
	Chopper_on AT %I* : BOOL;
	{attribute addProperty Name "Input_cycle_counter"}
	Input_cycle_counter AT %I* : BYTE;
	{attribute addProperty Name "DC_link_voltage"}
	DC_link_voltage AT %I* : UDINT;
	{attribute addProperty Name "Resistor_Current"}
	Resistor_Current AT %I* : DINT;
	{attribute addProperty Name "Duty_Cycle"}
	Duty_Cycle AT %I* : USINT;
END_STRUCT
END_TYPE

// ---- DUTs/IO/PDOs/BCT_Inputs_7ACE8FA6.TcDUT
{attribute 'GeneratedUsingTerminal: EJ9576-0000-0022'}
{attribute addProperty BoxType "EJ9576-0000-0022"}
{attribute addProperty Id "Terminal_OvertemperatureAT %I*BOOL1I2T_errorAT %I*BOOL1I2T_warningAT %I*BOOL1OvervoltageAT %I*BOOL1UndervoltageAT %I*BOOL1Chopper_onAT %I*BOOL1Overcurrent_ProtectionAT %I*BOOL1Input_cycle_counterAT %I*BYTE1DC_link_voltageAT %I*UDINT4Resistor_CurrentAT %I*DINT4Duty_CycleAT %I*USINT1"}
{attribute addProperty CRC "2060357542"}
{attribute addProperty Size "17"}
TYPE BCT_Inputs_7ACE8FA6 EXTENDS InputBase_8311D824 :
STRUCT
	{attribute addProperty Name "Terminal_Overtemperature"}
	Terminal_Overtemperature AT %I* : BOOL;
	{attribute addProperty Name "I2T_error"}
	I2T_error AT %I* : BOOL;
	{attribute addProperty Name "I2T_warning"}
	I2T_warning AT %I* : BOOL;
	{attribute addProperty Name "Overvoltage"}
	Overvoltage AT %I* : BOOL;
	{attribute addProperty Name "Undervoltage"}
	Undervoltage AT %I* : BOOL;
	{attribute addProperty Name "Chopper_on"}
	Chopper_on AT %I* : BOOL;
	{attribute addProperty Name "Overcurrent_Protection"}
	Overcurrent_Protection AT %I* : BOOL;
	{attribute addProperty Name "Input_cycle_counter"}
	Input_cycle_counter AT %I* : BYTE;
	{attribute addProperty Name "DC_link_voltage"}
	DC_link_voltage AT %I* : UDINT;
	{attribute addProperty Name "Resistor_Current"}
	Resistor_Current AT %I* : DINT;
	{attribute addProperty Name "Duty_Cycle"}
	Duty_Cycle AT %I* : USINT;
END_STRUCT
END_TYPE

// ---- DUTs/IO/PDOs/FSoE_Inputs_8952FEF0.TcDUT
{attribute 'GeneratedUsingTerminal: EJ1914-0000-0017'}
{attribute addProperty BoxType "EJ1914-0000-0017"}
{attribute addProperty Id "FSOEAT %I*FSOE_1F44E1B411"}
{attribute addProperty CRC "2303917808"}
{attribute addProperty Size "11"}
TYPE FSoE_Inputs_8952FEF0 EXTENDS InputBase_8311D824 :
STRUCT
	{attribute addProperty Name "FSOE"}
	FSOE AT %I* : FSOE_1F44E1B4;
END_STRUCT
END_TYPE

// ---- DUTs/IO/PDOs/FSoE_Outputs_7E672439.TcDUT
{attribute 'GeneratedUsingTerminal: EJ1914-0000-0017'}
{attribute addProperty BoxType "EJ1914-0000-0017"}
{attribute addProperty Id "FSOEAT %Q*FSOE_9A7ED3DD7"}
{attribute addProperty CRC "2120688697"}
{attribute addProperty Size "7"}
TYPE FSoE_Outputs_7E672439 EXTENDS OutputBase_10CEE7DE :
STRUCT
	{attribute addProperty Name "FSOE"}
	FSOE AT %Q* : FSOE_9A7ED3DD;
END_STRUCT
END_TYPE

// ---- DUTs/IO/PDOs/FIELDVOLTAGE_Field_Voltage_Status_9DC7C349.TcDUT
{attribute 'GeneratedUsingTerminal: EJ1914-0000-0017'}
{attribute addProperty BoxType "EJ1914-0000-0017"}
{attribute addProperty Id "Fieldvoltage_UnderrangeAT %I*BOOL1Fieldvoltage_OverrangeAT %I*BOOL1"}
{attribute addProperty CRC "2647114569"}
{attribute addProperty Size "2"}
TYPE FIELDVOLTAGE_Field_Voltage_Status_9DC7C349 EXTENDS InputBase_8311D824 :
STRUCT
	{attribute addProperty Name "Fieldvoltage_Underrange"}
	Fieldvoltage_Underrange AT %I* : BOOL;
	{attribute addProperty Name "Fieldvoltage_Overrange"}
	Fieldvoltage_Overrange AT %I* : BOOL;
END_STRUCT
END_TYPE

// ---- DUTs/IO/PDOs/FSLOGIC_Inputs_EEE9388E.TcDUT
{attribute 'GeneratedUsingTerminal: EJ1914-0000-0017'}
{attribute addProperty BoxType "EJ1914-0000-0017"}
{attribute addProperty Id "Safe_Logic_StateAT %I*USINT1Cycle_CounterAT %I*USINT1"}
{attribute addProperty CRC "4008261774"}
{attribute addProperty Size "2"}
TYPE FSLOGIC_Inputs_EEE9388E EXTENDS InputBase_8311D824 :
STRUCT
	{attribute addProperty Name "Safe_Logic_State"}
	Safe_Logic_State AT %I* : USINT;
	{attribute addProperty Name "Cycle_Counter"}
	Cycle_Counter AT %I* : USINT;
END_STRUCT
END_TYPE

// ---- DUTs/IO/PDOs/EMPTY_STRUCTURE.TcDUT
{attribute 'GeneratedUsingTerminal: EJ1914-0000-0017'}
{attribute addProperty BoxType "EJ1914-0000-0017"}
{attribute addProperty Id "EMPTY_STRUCTURE"}
{attribute addProperty CRC "0"}
{attribute addProperty Size "0"}
TYPE EMPTY_STRUCTURE :
STRUCT
END_STRUCT
END_TYPE

// ---- DUTs/IO/PDOs/Module_1_FSOE_5515F18A.TcDUT
{attribute 'GeneratedUsingTerminal: EJ1914-0000-0017'}
{attribute addProperty BoxType "EJ1914-0000-0017"}
{attribute addProperty Id "FSoE_InputsFSoE_Inputs_8952FEF011FSoE_OutputsFSoE_Outputs_7E6724397"}
{attribute addProperty CRC "1427501450"}
{attribute addProperty Size "18"}
TYPE Module_1_FSOE_5515F18A :
STRUCT
	{attribute addProperty Name "FSoE_Inputs"}
	FSoE_Inputs  : FSoE_Inputs_8952FEF0;
	{attribute addProperty Name "FSoE_Outputs"}
	FSoE_Outputs  : FSoE_Outputs_7E672439;
END_STRUCT
END_TYPE

// ---- DUTs/IO/PDOs/Module_2_DEVICEIO_5FA6B4E7.TcDUT
{attribute 'GeneratedUsingTerminal: EJ1914-0000-0017'}
{attribute addProperty BoxType "EJ1914-0000-0017"}
{attribute addProperty Id "FIELDVOLTAGE_Field_Voltage_StatusFIELDVOLTAGE_Field_Voltage_Status_9DC7C3492"}
{attribute addProperty CRC "1604760807"}
{attribute addProperty Size "2"}
TYPE Module_2_DEVICEIO_5FA6B4E7 :
STRUCT
	{attribute addProperty Name "FIELDVOLTAGE_Field_Voltage_Status"}
	FIELDVOLTAGE_Field_Voltage_Status  : FIELDVOLTAGE_Field_Voltage_Status_9DC7C349;
END_STRUCT
END_TYPE

// ---- DUTs/IO/PDOs/Module_3_FSLOGIC_DEAB4522.TcDUT
{attribute 'GeneratedUsingTerminal: EJ1914-0000-0017'}
{attribute addProperty BoxType "EJ1914-0000-0017"}
{attribute addProperty Id "FSLOGIC_InputsFSLOGIC_Inputs_EEE9388E2FSLOGIC_OutputsEMPTY_STRUCTURE0"}
{attribute addProperty CRC "3735766306"}
{attribute addProperty Size "2"}
TYPE Module_3_FSLOGIC_DEAB4522 :
STRUCT
	{attribute addProperty Name "FSLOGIC_Inputs"}
	FSLOGIC_Inputs  : FSLOGIC_Inputs_EEE9388E;
	{attribute addProperty Name "FSLOGIC_Outputs"}
	FSLOGIC_Outputs  : EMPTY_STRUCTURE;
END_STRUCT
END_TYPE

// ---- DUTs/IO/PDOs/FSoE_Inputs_C661B78A.TcDUT
{attribute 'GeneratedUsingTerminal: EJ1918-0000-0017'}
{attribute addProperty BoxType "EJ1918-0000-0017"}
{attribute addProperty Id "FSOEAT %I*FSOE_9F04885D17"}
{attribute addProperty CRC "3328292746"}
{attribute addProperty Size "17"}
TYPE FSoE_Inputs_C661B78A EXTENDS InputBase_8311D824 :
STRUCT
	{attribute addProperty Name "FSOE"}
	FSOE AT %I* : FSOE_9F04885D;
END_STRUCT
END_TYPE

// ---- DUTs/IO/PDOs/FSoE_Outputs_E138FCB5.TcDUT
{attribute 'GeneratedUsingTerminal: EJ1918-0000-0017'}
{attribute addProperty BoxType "EJ1918-0000-0017"}
{attribute addProperty Id "FSOEAT %Q*FSOE_878484619"}
{attribute addProperty CRC "3778608309"}
{attribute addProperty Size "9"}
TYPE FSoE_Outputs_E138FCB5 EXTENDS OutputBase_10CEE7DE :
STRUCT
	{attribute addProperty Name "FSOE"}
	FSOE AT %Q* : FSOE_87848461;
END_STRUCT
END_TYPE

// ---- DUTs/IO/PDOs/Module_1_FSOE_18ED951F.TcDUT
{attribute 'GeneratedUsingTerminal: EJ1918-0000-0017'}
{attribute addProperty BoxType "EJ1918-0000-0017"}
{attribute addProperty Id "FSoE_InputsFSoE_Inputs_C661B78A17FSoE_OutputsFSoE_Outputs_E138FCB59"}
{attribute addProperty CRC "418223391"}
{attribute addProperty Size "26"}
TYPE Module_1_FSOE_18ED951F :
STRUCT
	{attribute addProperty Name "FSoE_Inputs"}
	FSoE_Inputs  : FSoE_Inputs_C661B78A;
	{attribute addProperty Name "FSoE_Outputs"}
	FSoE_Outputs  : FSoE_Outputs_E138FCB5;
END_STRUCT
END_TYPE

// ---- DUTs/IO/PDOs/FSoE_Inputs_8A5FBAF8.TcDUT
{attribute 'GeneratedUsingTerminal: EJ1957-0000-0017'}
{attribute addProperty BoxType "EJ1957-0000-0017"}
{attribute addProperty Id "FSOEAT %I*FSOE_BBC930F718"}
{attribute addProperty CRC "2321529592"}
{attribute addProperty Size "18"}
TYPE FSoE_Inputs_8A5FBAF8 EXTENDS InputBase_8311D824 :
STRUCT
	{attribute addProperty Name "FSOE"}
	FSOE AT %I* : FSOE_BBC930F7;
END_STRUCT
END_TYPE

// ---- DUTs/IO/PDOs/FSoE_Outputs_1F40D103.TcDUT
{attribute 'GeneratedUsingTerminal: EJ1957-0000-0017'}
{attribute addProperty BoxType "EJ1957-0000-0017"}
{attribute addProperty Id "FSOEAT %Q*FSOE_D1C9D1EA14"}
{attribute addProperty CRC "524341507"}
{attribute addProperty Size "14"}
TYPE FSoE_Outputs_1F40D103 EXTENDS OutputBase_10CEE7DE :
STRUCT
	{attribute addProperty Name "FSOE"}
	FSOE AT %Q* : FSOE_D1C9D1EA;
END_STRUCT
END_TYPE

// ---- DUTs/IO/PDOs/Outputs_7EDA7A42.TcDUT
{attribute 'GeneratedUsingTerminal: EJ1957-0000-0017'}
{attribute addProperty BoxType "EJ1957-0000-0017"}
{attribute addProperty Id "Channel_1_Standard_OutputAT %Q*BOOL1Channel_2_Standard_OutputAT %Q*BOOL1Channel_3_Standard_OutputAT %Q*BOOL1Channel_4_Standard_OutputAT %Q*BOOL1"}
{attribute addProperty CRC "2128247362"}
{attribute addProperty Size "4"}
TYPE Outputs_7EDA7A42 EXTENDS OutputBase_10CEE7DE :
STRUCT
	{attribute addProperty Name "Channel_1_Standard_Output"}
	Channel_1_Standard_Output AT %Q* : BOOL;
	{attribute addProperty Name "Channel_2_Standard_Output"}
	Channel_2_Standard_Output AT %Q* : BOOL;
	{attribute addProperty Name "Channel_3_Standard_Output"}
	Channel_3_Standard_Output AT %Q* : BOOL;
	{attribute addProperty Name "Channel_4_Standard_Output"}
	Channel_4_Standard_Output AT %Q* : BOOL;
END_STRUCT
END_TYPE

// ---- DUTs/IO/PDOs/WcState_B516A264.TcDUT
{attribute 'GeneratedUsingTerminal: EJ1957-0000-0017'}
{attribute addProperty BoxType "EJ1957-0000-0017"}
{attribute addProperty Id "WcState0AT %I*BOOL1WcState1AT %I*BOOL1InputToggle0AT %I*BOOL1InputToggle1AT %I*BOOL1"}
{attribute addProperty CRC "3038159460"}
{attribute addProperty Size "4"}
TYPE WcState_B516A264 EXTENDS InputBase_8311D824 :
STRUCT
	{attribute addProperty Name "WcState0"}
	WcState0 AT %I* : BOOL;
	{attribute addProperty Name "WcState1"}
	WcState1 AT %I* : BOOL;
	{attribute addProperty Name "InputToggle0"}
	InputToggle0 AT %I* : BOOL;
	{attribute addProperty Name "InputToggle1"}
	InputToggle1 AT %I* : BOOL;
END_STRUCT
END_TYPE

// ---- DUTs/IO/PDOs/Module_1_FSOE_9FCACE14.TcDUT
{attribute 'GeneratedUsingTerminal: EJ1957-0000-0017'}
{attribute addProperty BoxType "EJ1957-0000-0017"}
{attribute addProperty Id "FSoE_InputsFSoE_Inputs_8A5FBAF818FSoE_OutputsFSoE_Outputs_1F40D10314"}
{attribute addProperty CRC "2680868372"}
{attribute addProperty Size "32"}
TYPE Module_1_FSOE_9FCACE14 :
STRUCT
	{attribute addProperty Name "FSoE_Inputs"}
	FSoE_Inputs  : FSoE_Inputs_8A5FBAF8;
	{attribute addProperty Name "FSoE_Outputs"}
	FSoE_Outputs  : FSoE_Outputs_1F40D103;
END_STRUCT
END_TYPE

// ---- DUTs/IO/PDOs/Module_2_FSOUT_5A5AEBA4.TcDUT
{attribute 'GeneratedUsingTerminal: EJ1957-0000-0017'}
{attribute addProperty BoxType "EJ1957-0000-0017"}
{attribute addProperty Id "OutputsOutputs_7EDA7A424"}
{attribute addProperty CRC "1515908004"}
{attribute addProperty Size "4"}
TYPE Module_2_FSOUT_5A5AEBA4 :
STRUCT
	{attribute addProperty Name "Outputs"}
	Outputs  : Outputs_7EDA7A42;
END_STRUCT
END_TYPE

// ---- DUTs/IO/PDOs/Module_3_DEVICEIO_5FA6B4E7.TcDUT
{attribute 'GeneratedUsingTerminal: EJ1957-0000-0017'}
{attribute addProperty BoxType "EJ1957-0000-0017"}
{attribute addProperty Id "FIELDVOLTAGE_Field_Voltage_StatusFIELDVOLTAGE_Field_Voltage_Status_9DC7C3492"}
{attribute addProperty CRC "1604760807"}
{attribute addProperty Size "2"}
TYPE Module_3_DEVICEIO_5FA6B4E7 :
STRUCT
	{attribute addProperty Name "FIELDVOLTAGE_Field_Voltage_Status"}
	FIELDVOLTAGE_Field_Voltage_Status  : FIELDVOLTAGE_Field_Voltage_Status_9DC7C349;
END_STRUCT
END_TYPE

// ---- DUTs/IO/PDOs/Module_4_FSLOGIC_DEAB4522.TcDUT
{attribute 'GeneratedUsingTerminal: EJ1957-0000-0017'}
{attribute addProperty BoxType "EJ1957-0000-0017"}
{attribute addProperty Id "FSLOGIC_InputsFSLOGIC_Inputs_EEE9388E2FSLOGIC_OutputsEMPTY_STRUCTURE0"}
{attribute addProperty CRC "3735766306"}
{attribute addProperty Size "2"}
TYPE Module_4_FSLOGIC_DEAB4522 :
STRUCT
	{attribute addProperty Name "FSLOGIC_Inputs"}
	FSLOGIC_Inputs  : FSLOGIC_Inputs_EEE9388E;
	{attribute addProperty Name "FSLOGIC_Outputs"}
	FSLOGIC_Outputs  : EMPTY_STRUCTURE;
END_STRUCT
END_TYPE

// ---- DUTs/IO/PDOs/FSoE_Inputs_15C2E7B1.TcDUT
{attribute 'GeneratedUsingTerminal: EJ2914-0000-0017'}
{attribute addProperty BoxType "EJ2914-0000-0017"}
{attribute addProperty Id "FSOEAT %I*FSOE_D94E700C6"}
{attribute addProperty CRC "365094833"}
{attribute addProperty Size "6"}
TYPE FSoE_Inputs_15C2E7B1 EXTENDS InputBase_8311D824 :
STRUCT
	{attribute addProperty Name "FSOE"}
	FSOE AT %I* : FSOE_D94E700C;
END_STRUCT
END_TYPE

// ---- DUTs/IO/PDOs/FSoE_Outputs_C9D9BEFD.TcDUT
{attribute 'GeneratedUsingTerminal: EJ2914-0000-0017'}
{attribute addProperty BoxType "EJ2914-0000-0017"}
{attribute addProperty Id "FSOEAT %Q*FSOE_1DB604F410"}
{attribute addProperty CRC "3386490621"}
{attribute addProperty Size "10"}
TYPE FSoE_Outputs_C9D9BEFD EXTENDS OutputBase_10CEE7DE :
STRUCT
	{attribute addProperty Name "FSOE"}
	FSOE AT %Q* : FSOE_1DB604F4;
END_STRUCT
END_TYPE

// ---- DUTs/IO/PDOs/Module_1_FSOE_212A0B66.TcDUT
{attribute 'GeneratedUsingTerminal: EJ2914-0000-0017'}
{attribute addProperty BoxType "EJ2914-0000-0017"}
{attribute addProperty Id "FSoE_InputsFSoE_Inputs_15C2E7B16FSoE_OutputsFSoE_Outputs_C9D9BEFD10"}
{attribute addProperty CRC "556403558"}
{attribute addProperty Size "16"}
TYPE Module_1_FSOE_212A0B66 :
STRUCT
	{attribute addProperty Name "FSoE_Inputs"}
	FSoE_Inputs  : FSoE_Inputs_15C2E7B1;
	{attribute addProperty Name "FSoE_Outputs"}
	FSoE_Outputs  : FSoE_Outputs_C9D9BEFD;
END_STRUCT
END_TYPE

// ---- DUTs/IO/PDOs/FSoE_Inputs_939ABF3D.TcDUT
{attribute 'GeneratedUsingTerminal: EJ2918-0000-0017'}
{attribute addProperty BoxType "EJ2918-0000-0017"}
{attribute addProperty Id "FSOEAT %I*FSOE_046F804E7"}
{attribute addProperty CRC "2476392253"}
{attribute addProperty Size "7"}
TYPE FSoE_Inputs_939ABF3D EXTENDS InputBase_8311D824 :
STRUCT
	{attribute addProperty Name "FSOE"}
	FSOE AT %I* : FSOE_046F804E;
END_STRUCT
END_TYPE

// ---- DUTs/IO/PDOs/FSoE_Outputs_2DD09AA7.TcDUT
{attribute 'GeneratedUsingTerminal: EJ2918-0000-0017'}
{attribute addProperty BoxType "EJ2918-0000-0017"}
{attribute addProperty Id "FSOEAT %Q*FSOE_2DC96D3115"}
{attribute addProperty CRC "768645799"}
{attribute addProperty Size "15"}
TYPE FSoE_Outputs_2DD09AA7 EXTENDS OutputBase_10CEE7DE :
STRUCT
	{attribute addProperty Name "FSOE"}
	FSOE AT %Q* : FSOE_2DC96D31;
END_STRUCT
END_TYPE

// ---- DUTs/IO/PDOs/Outputs_FB9F3520.TcDUT
{attribute 'GeneratedUsingTerminal: EJ2918-0000-0017'}
{attribute addProperty BoxType "EJ2918-0000-0017"}
{attribute addProperty Id "Module_1_Channel_1_Standard_OutputAT %Q*BOOL1Module_1_Channel_2_Standard_OutputAT %Q*BOOL1Module_1_Channel_3_Standard_OutputAT %Q*BOOL1Module_1_Channel_4_Standard_OutputAT %Q*BOOL1Module_2_Channel_1_Standard_OutputAT %Q*BOOL1Module_2_Channel_2_Standard_OutputAT %Q*BOOL1Module_2_Channel_3_Standard_OutputAT %Q*BOOL1Module_2_Channel_4_Standard_OutputAT %Q*BOOL1"}
{attribute addProperty CRC "4221515040"}
{attribute addProperty Size "8"}
TYPE Outputs_FB9F3520 EXTENDS OutputBase_10CEE7DE :
STRUCT
	{attribute addProperty Name "Module_1_Channel_1_Standard_Output"}
	Module_1_Channel_1_Standard_Output AT %Q* : BOOL;
	{attribute addProperty Name "Module_1_Channel_2_Standard_Output"}
	Module_1_Channel_2_Standard_Output AT %Q* : BOOL;
	{attribute addProperty Name "Module_1_Channel_3_Standard_Output"}
	Module_1_Channel_3_Standard_Output AT %Q* : BOOL;
	{attribute addProperty Name "Module_1_Channel_4_Standard_Output"}
	Module_1_Channel_4_Standard_Output AT %Q* : BOOL;
	{attribute addProperty Name "Module_2_Channel_1_Standard_Output"}
	Module_2_Channel_1_Standard_Output AT %Q* : BOOL;
	{attribute addProperty Name "Module_2_Channel_2_Standard_Output"}
	Module_2_Channel_2_Standard_Output AT %Q* : BOOL;
	{attribute addProperty Name "Module_2_Channel_3_Standard_Output"}
	Module_2_Channel_3_Standard_Output AT %Q* : BOOL;
	{attribute addProperty Name "Module_2_Channel_4_Standard_Output"}
	Module_2_Channel_4_Standard_Output AT %Q* : BOOL;
END_STRUCT
END_TYPE

// ---- DUTs/IO/PDOs/Module_1_FSOE_7F12D292.TcDUT
{attribute 'GeneratedUsingTerminal: EJ2918-0000-0017'}
{attribute addProperty BoxType "EJ2918-0000-0017"}
{attribute addProperty Id "FSoE_InputsFSoE_Inputs_939ABF3D7FSoE_OutputsFSoE_Outputs_2DD09AA715"}
{attribute addProperty CRC "2131939986"}
{attribute addProperty Size "22"}
TYPE Module_1_FSOE_7F12D292 :
STRUCT
	{attribute addProperty Name "FSoE_Inputs"}
	FSoE_Inputs  : FSoE_Inputs_939ABF3D;
	{attribute addProperty Name "FSoE_Outputs"}
	FSoE_Outputs  : FSoE_Outputs_2DD09AA7;
END_STRUCT
END_TYPE

// ---- DUTs/IO/PDOs/Module_2_FSOUT_9813A38E.TcDUT
{attribute 'GeneratedUsingTerminal: EJ2918-0000-0017'}
{attribute addProperty BoxType "EJ2918-0000-0017"}
{attribute addProperty Id "OutputsOutputs_FB9F35208"}
{attribute addProperty CRC "2551423886"}
{attribute addProperty Size "8"}
TYPE Module_2_FSOUT_9813A38E :
STRUCT
	{attribute addProperty Name "Outputs"}
	Outputs  : Outputs_FB9F3520;
END_STRUCT
END_TYPE

// ---- DUTs/IO/PDOs/InfoData_E68C61CD.TcDUT
{attribute 'GeneratedUsingTerminal: IODEVICETYPE_ETHERCATPROT'}
{attribute addProperty BoxType "IODEVICETYPE_ETHERCATPROT"}
{attribute addProperty Id "ChangeCountAT %I*UINT2DevIdAT %I*UINT2AmsNetIdAT %I*AMSNETID6CfgSlaveCountAT %I*UINT2DcToTcTimeOffsetAT %I*LINT8DcToExtTimeOffsetAT %I*LINT8"}
{attribute addProperty CRC "3867959757"}
{attribute addProperty Size "28"}
TYPE InfoData_E68C61CD EXTENDS InputBase_8311D824 :
STRUCT
	{attribute addProperty Name "ChangeCount"}
	ChangeCount AT %I* : UINT;
	{attribute addProperty Name "DevId"}
	DevId AT %I* : UINT;
	{attribute addProperty Name "AmsNetId"}
	AmsNetId AT %I* : AMSNETID;
	{attribute addProperty Name "CfgSlaveCount"}
	CfgSlaveCount AT %I* : UINT;
	{attribute addProperty Name "DcToTcTimeOffset"}
	DcToTcTimeOffset AT %I* : LINT;
	{attribute addProperty Name "DcToExtTimeOffset"}
	DcToExtTimeOffset AT %I* : LINT;
END_STRUCT
END_TYPE

// ---- DUTs/IO/PDOs/InfoData_2A97D6CF.TcDUT
{attribute 'GeneratedUsingTerminal: IODEVICETYPE_ETHERCATPROT'}
{attribute addProperty BoxType "IODEVICETYPE_ETHERCATPROT"}
{attribute addProperty Id "ObjectIdAT %I*OTCID4StateAT %I*UINT2SlaveCountAT %I*UINT2"}
{attribute addProperty CRC "714593999"}
{attribute addProperty Size "8"}
TYPE InfoData_2A97D6CF EXTENDS InputBase_8311D824 :
STRUCT
	{attribute addProperty Name "ObjectId"}
	ObjectId AT %I* : OTCID;
	{attribute addProperty Name "State"}
	State AT %I* : UINT;
	{attribute addProperty Name "SlaveCount"}
	SlaveCount AT %I* : UINT;
END_STRUCT
END_TYPE

// ---- DUTs/IO/PDOs/Inputs_25A0042B.TcDUT
{attribute 'GeneratedUsingTerminal: IODEVICETYPE_ETHERCATPROT'}
{attribute addProperty BoxType "IODEVICETYPE_ETHERCATPROT"}
{attribute addProperty Id "SlaveCountAT %I*UINT2DevStateAT %I*UINT2Frm0StateAT %I*UINT2Frm0WcStateAT %I*UINT2Frm0InputToggleAT %I*UINT2Frm1StateAT %I*UINT2Frm1WcStateAT %I*UINT2Frm1InputToggleAT %I*UINT2Frm2StateAT %I*UINT2Frm2WcStateAT %I*UINT2Frm2InputToggleAT %I*UINT2Frm3StateAT %I*UINT2Frm3WcStateAT %I*UINT2Frm3InputToggleAT %I*UINT2Frm4StateAT %I*UINT2Frm4WcStateAT %I*UINT2Frm4InputToggleAT %I*UINT2Frm5StateAT %I*UINT2Frm5WcStateAT %I*UINT2Frm5InputToggleAT %I*UINT2Frm6StateAT %I*UINT2Frm6WcStateAT %I*UINT2Frm6InputToggleAT %I*UINT2Frm7StateAT %I*UINT2Frm7WcStateAT %I*UINT2Frm7InputToggleAT %I*UINT2Frm8StateAT %I*UINT2Frm8WcStateAT %I*UINT2Frm8InputToggleAT %I*UINT2Frm9StateAT %I*UINT2Frm9WcStateAT %I*UINT2Frm9InputToggleAT %I*UINT2Frm10StateAT %I*UINT2Frm10WcStateAT %I*UINT2Frm10InputToggleAT %I*UINT2Frm11StateAT %I*UINT2Frm11WcStateAT %I*UINT2Frm11InputToggleAT %I*UINT2Frm12StateAT %I*UINT2Frm12WcStateAT %I*UINT2Frm12InputToggleAT %I*UINT2Frm13StateAT %I*UINT2Frm13WcStateAT %I*UINT2Frm13InputToggleAT %I*UINT2Frm14StateAT %I*UINT2Frm14WcStateAT %I*UINT2Frm14InputToggleAT %I*UINT2Frm15StateAT %I*UINT2Frm15WcStateAT %I*UINT2Frm15InputToggleAT %I*UINT2Frm16StateAT %I*UINT2Frm16WcStateAT %I*UINT2Frm16InputToggleAT %I*UINT2Frm17StateAT %I*UINT2Frm17WcStateAT %I*UINT2Frm17InputToggleAT %I*UINT2Frm18StateAT %I*UINT2Frm18WcStateAT %I*UINT2Frm18InputToggleAT %I*UINT2Frm19StateAT %I*UINT2Frm19WcStateAT %I*UINT2Frm19InputToggleAT %I*UINT2Frm20StateAT %I*UINT2Frm20WcStateAT %I*UINT2Frm20InputToggleAT %I*UINT2Frm21StateAT %I*UINT2Frm21WcStateAT %I*UINT2Frm21InputToggleAT %I*UINT2Frm22StateAT %I*UINT2Frm22WcStateAT %I*UINT2Frm22InputToggleAT %I*UINT2Frm23StateAT %I*UINT2Frm23WcStateAT %I*UINT2Frm23InputToggleAT %I*UINT2Frm24StateAT %I*UINT2Frm24WcStateAT %I*UINT2Frm24InputToggleAT %I*UINT2Frm25StateAT %I*UINT2Frm25WcStateAT %I*UINT2Frm25InputToggleAT %I*UINT2"}
{attribute addProperty CRC "631243819"}
{attribute addProperty Size "160"}
TYPE Inputs_25A0042B EXTENDS InputBase_8311D824 :
STRUCT
	{attribute addProperty Name "SlaveCount"}
	SlaveCount AT %I* : UINT;
	{attribute addProperty Name "DevState"}
	DevState AT %I* : UINT;
	{attribute addProperty Name "Frm0State"}
	Frm0State AT %I* : UINT;
	{attribute addProperty Name "Frm0WcState"}
	Frm0WcState AT %I* : UINT;
	{attribute addProperty Name "Frm0InputToggle"}
	Frm0InputToggle AT %I* : UINT;
	{attribute addProperty Name "Frm1State"}
	Frm1State AT %I* : UINT;
	{attribute addProperty Name "Frm1WcState"}
	Frm1WcState AT %I* : UINT;
	{attribute addProperty Name "Frm1InputToggle"}
	Frm1InputToggle AT %I* : UINT;
	{attribute addProperty Name "Frm2State"}
	Frm2State AT %I* : UINT;
	{attribute addProperty Name "Frm2WcState"}
	Frm2WcState AT %I* : UINT;
	{attribute addProperty Name "Frm2InputToggle"}
	Frm2InputToggle AT %I* : UINT;
	{attribute addProperty Name "Frm3State"}
	Frm3State AT %I* : UINT;
	{attribute addProperty Name "Frm3WcState"}
	Frm3WcState AT %I* : UINT;
	{attribute addProperty Name "Frm3InputToggle"}
	Frm3InputToggle AT %I* : UINT;
	{attribute addProperty Name "Frm4State"}
	Frm4State AT %I* : UINT;
	{attribute addProperty Name "Frm4WcState"}
	Frm4WcState AT %I* : UINT;
	{attribute addProperty Name "Frm4InputToggle"}
	Frm4InputToggle AT %I* : UINT;
	{attribute addProperty Name "Frm5State"}
	Frm5State AT %I* : UINT;
	{attribute addProperty Name "Frm5WcState"}
	Frm5WcState AT %I* : UINT;
	{attribute addProperty Name "Frm5InputToggle"}
	Frm5InputToggle AT %I* : UINT;
	{attribute addProperty Name "Frm6State"}
	Frm6State AT %I* : UINT;
	{attribute addProperty Name "Frm6WcState"}
	Frm6WcState AT %I* : UINT;
	{attribute addProperty Name "Frm6InputToggle"}
	Frm6InputToggle AT %I* : UINT;
	{attribute addProperty Name "Frm7State"}
	Frm7State AT %I* : UINT;
	{attribute addProperty Name "Frm7WcState"}
	Frm7WcState AT %I* : UINT;
	{attribute addProperty Name "Frm7InputToggle"}
	Frm7InputToggle AT %I* : UINT;
	{attribute addProperty Name "Frm8State"}
	Frm8State AT %I* : UINT;
	{attribute addProperty Name "Frm8WcState"}
	Frm8WcState AT %I* : UINT;
	{attribute addProperty Name "Frm8InputToggle"}
	Frm8InputToggle AT %I* : UINT;
	{attribute addProperty Name "Frm9State"}
	Frm9State AT %I* : UINT;
	{attribute addProperty Name "Frm9WcState"}
	Frm9WcState AT %I* : UINT;
	{attribute addProperty Name "Frm9InputToggle"}
	Frm9InputToggle AT %I* : UINT;
	{attribute addProperty Name "Frm10State"}
	Frm10State AT %I* : UINT;
	{attribute addProperty Name "Frm10WcState"}
	Frm10WcState AT %I* : UINT;
	{attribute addProperty Name "Frm10InputToggle"}
	Frm10InputToggle AT %I* : UINT;
	{attribute addProperty Name "Frm11State"}
	Frm11State AT %I* : UINT;
	{attribute addProperty Name "Frm11WcState"}
	Frm11WcState AT %I* : UINT;
	{attribute addProperty Name "Frm11InputToggle"}
	Frm11InputToggle AT %I* : UINT;
	{attribute addProperty Name "Frm12State"}
	Frm12State AT %I* : UINT;
	{attribute addProperty Name "Frm12WcState"}
	Frm12WcState AT %I* : UINT;
	{attribute addProperty Name "Frm12InputToggle"}
	Frm12InputToggle AT %I* : UINT;
	{attribute addProperty Name "Frm13State"}
	Frm13State AT %I* : UINT;
	{attribute addProperty Name "Frm13WcState"}
	Frm13WcState AT %I* : UINT;
	{attribute addProperty Name "Frm13InputToggle"}
	Frm13InputToggle AT %I* : UINT;
	{attribute addProperty Name "Frm14State"}
	Frm14State AT %I* : UINT;
	{attribute addProperty Name "Frm14WcState"}
	Frm14WcState AT %I* : UINT;
	{attribute addProperty Name "Frm14InputToggle"}
	Frm14InputToggle AT %I* : UINT;
	{attribute addProperty Name "Frm15State"}
	Frm15State AT %I* : UINT;
	{attribute addProperty Name "Frm15WcState"}
	Frm15WcState AT %I* : UINT;
	{attribute addProperty Name "Frm15InputToggle"}
	Frm15InputToggle AT %I* : UINT;
	{attribute addProperty Name "Frm16State"}
	Frm16State AT %I* : UINT;
	{attribute addProperty Name "Frm16WcState"}
	Frm16WcState AT %I* : UINT;
	{attribute addProperty Name "Frm16InputToggle"}
	Frm16InputToggle AT %I* : UINT;
	{attribute addProperty Name "Frm17State"}
	Frm17State AT %I* : UINT;
	{attribute addProperty Name "Frm17WcState"}
	Frm17WcState AT %I* : UINT;
	{attribute addProperty Name "Frm17InputToggle"}
	Frm17InputToggle AT %I* : UINT;
	{attribute addProperty Name "Frm18State"}
	Frm18State AT %I* : UINT;
	{attribute addProperty Name "Frm18WcState"}
	Frm18WcState AT %I* : UINT;
	{attribute addProperty Name "Frm18InputToggle"}
	Frm18InputToggle AT %I* : UINT;
	{attribute addProperty Name "Frm19State"}
	Frm19State AT %I* : UINT;
	{attribute addProperty Name "Frm19WcState"}
	Frm19WcState AT %I* : UINT;
	{attribute addProperty Name "Frm19InputToggle"}
	Frm19InputToggle AT %I* : UINT;
	{attribute addProperty Name "Frm20State"}
	Frm20State AT %I* : UINT;
	{attribute addProperty Name "Frm20WcState"}
	Frm20WcState AT %I* : UINT;
	{attribute addProperty Name "Frm20InputToggle"}
	Frm20InputToggle AT %I* : UINT;
	{attribute addProperty Name "Frm21State"}
	Frm21State AT %I* : UINT;
	{attribute addProperty Name "Frm21WcState"}
	Frm21WcState AT %I* : UINT;
	{attribute addProperty Name "Frm21InputToggle"}
	Frm21InputToggle AT %I* : UINT;
	{attribute addProperty Name "Frm22State"}
	Frm22State AT %I* : UINT;
	{attribute addProperty Name "Frm22WcState"}
	Frm22WcState AT %I* : UINT;
	{attribute addProperty Name "Frm22InputToggle"}
	Frm22InputToggle AT %I* : UINT;
	{attribute addProperty Name "Frm23State"}
	Frm23State AT %I* : UINT;
	{attribute addProperty Name "Frm23WcState"}
	Frm23WcState AT %I* : UINT;
	{attribute addProperty Name "Frm23InputToggle"}
	Frm23InputToggle AT %I* : UINT;
	{attribute addProperty Name "Frm24State"}
	Frm24State AT %I* : UINT;
	{attribute addProperty Name "Frm24WcState"}
	Frm24WcState AT %I* : UINT;
	{attribute addProperty Name "Frm24InputToggle"}
	Frm24InputToggle AT %I* : UINT;
	{attribute addProperty Name "Frm25State"}
	Frm25State AT %I* : UINT;
	{attribute addProperty Name "Frm25WcState"}
	Frm25WcState AT %I* : UINT;
	{attribute addProperty Name "Frm25InputToggle"}
	Frm25InputToggle AT %I* : UINT;
END_STRUCT
END_TYPE

// ---- DUTs/IO/PDOs/Outputs_2397A10E.TcDUT
{attribute 'GeneratedUsingTerminal: IODEVICETYPE_ETHERCATPROT'}
{attribute addProperty BoxType "IODEVICETYPE_ETHERCATPROT"}
{attribute addProperty Id "DevCtrlAT %Q*UINT2Frm0CtrlAT %Q*UINT2Frm0WcCtrlAT %Q*UINT2Frm1CtrlAT %Q*UINT2Frm1WcCtrlAT %Q*UINT2Frm2CtrlAT %Q*UINT2Frm2WcCtrlAT %Q*UINT2Frm3CtrlAT %Q*UINT2Frm3WcCtrlAT %Q*UINT2Frm4CtrlAT %Q*UINT2Frm4WcCtrlAT %Q*UINT2Frm5CtrlAT %Q*UINT2Frm5WcCtrlAT %Q*UINT2Frm6CtrlAT %Q*UINT2Frm6WcCtrlAT %Q*UINT2Frm7CtrlAT %Q*UINT2Frm7WcCtrlAT %Q*UINT2Frm8CtrlAT %Q*UINT2Frm8WcCtrlAT %Q*UINT2Frm9CtrlAT %Q*UINT2Frm9WcCtrlAT %Q*UINT2Frm10CtrlAT %Q*UINT2Frm10WcCtrlAT %Q*UINT2Frm11CtrlAT %Q*UINT2Frm11WcCtrlAT %Q*UINT2Frm12CtrlAT %Q*UINT2Frm12WcCtrlAT %Q*UINT2Frm13CtrlAT %Q*UINT2Frm13WcCtrlAT %Q*UINT2Frm14CtrlAT %Q*UINT2Frm14WcCtrlAT %Q*UINT2Frm15CtrlAT %Q*UINT2Frm15WcCtrlAT %Q*UINT2Frm16CtrlAT %Q*UINT2Frm16WcCtrlAT %Q*UINT2Frm17CtrlAT %Q*UINT2Frm17WcCtrlAT %Q*UINT2Frm18CtrlAT %Q*UINT2Frm18WcCtrlAT %Q*UINT2Frm19CtrlAT %Q*UINT2Frm19WcCtrlAT %Q*UINT2Frm20CtrlAT %Q*UINT2Frm20WcCtrlAT %Q*UINT2Frm21CtrlAT %Q*UINT2Frm21WcCtrlAT %Q*UINT2Frm22CtrlAT %Q*UINT2Frm22WcCtrlAT %Q*UINT2Frm23CtrlAT %Q*UINT2Frm23WcCtrlAT %Q*UINT2Frm24CtrlAT %Q*UINT2Frm24WcCtrlAT %Q*UINT2Frm25CtrlAT %Q*UINT2Frm25WcCtrlAT %Q*UINT2"}
{attribute addProperty CRC "597139726"}
{attribute addProperty Size "106"}
TYPE Outputs_2397A10E EXTENDS OutputBase_10CEE7DE :
STRUCT
	{attribute addProperty Name "DevCtrl"}
	DevCtrl AT %Q* : UINT;
	{attribute addProperty Name "Frm0Ctrl"}
	Frm0Ctrl AT %Q* : UINT;
	{attribute addProperty Name "Frm0WcCtrl"}
	Frm0WcCtrl AT %Q* : UINT;
	{attribute addProperty Name "Frm1Ctrl"}
	Frm1Ctrl AT %Q* : UINT;
	{attribute addProperty Name "Frm1WcCtrl"}
	Frm1WcCtrl AT %Q* : UINT;
	{attribute addProperty Name "Frm2Ctrl"}
	Frm2Ctrl AT %Q* : UINT;
	{attribute addProperty Name "Frm2WcCtrl"}
	Frm2WcCtrl AT %Q* : UINT;
	{attribute addProperty Name "Frm3Ctrl"}
	Frm3Ctrl AT %Q* : UINT;
	{attribute addProperty Name "Frm3WcCtrl"}
	Frm3WcCtrl AT %Q* : UINT;
	{attribute addProperty Name "Frm4Ctrl"}
	Frm4Ctrl AT %Q* : UINT;
	{attribute addProperty Name "Frm4WcCtrl"}
	Frm4WcCtrl AT %Q* : UINT;
	{attribute addProperty Name "Frm5Ctrl"}
	Frm5Ctrl AT %Q* : UINT;
	{attribute addProperty Name "Frm5WcCtrl"}
	Frm5WcCtrl AT %Q* : UINT;
	{attribute addProperty Name "Frm6Ctrl"}
	Frm6Ctrl AT %Q* : UINT;
	{attribute addProperty Name "Frm6WcCtrl"}
	Frm6WcCtrl AT %Q* : UINT;
	{attribute addProperty Name "Frm7Ctrl"}
	Frm7Ctrl AT %Q* : UINT;
	{attribute addProperty Name "Frm7WcCtrl"}
	Frm7WcCtrl AT %Q* : UINT;
	{attribute addProperty Name "Frm8Ctrl"}
	Frm8Ctrl AT %Q* : UINT;
	{attribute addProperty Name "Frm8WcCtrl"}
	Frm8WcCtrl AT %Q* : UINT;
	{attribute addProperty Name "Frm9Ctrl"}
	Frm9Ctrl AT %Q* : UINT;
	{attribute addProperty Name "Frm9WcCtrl"}
	Frm9WcCtrl AT %Q* : UINT;
	{attribute addProperty Name "Frm10Ctrl"}
	Frm10Ctrl AT %Q* : UINT;
	{attribute addProperty Name "Frm10WcCtrl"}
	Frm10WcCtrl AT %Q* : UINT;
	{attribute addProperty Name "Frm11Ctrl"}
	Frm11Ctrl AT %Q* : UINT;
	{attribute addProperty Name "Frm11WcCtrl"}
	Frm11WcCtrl AT %Q* : UINT;
	{attribute addProperty Name "Frm12Ctrl"}
	Frm12Ctrl AT %Q* : UINT;
	{attribute addProperty Name "Frm12WcCtrl"}
	Frm12WcCtrl AT %Q* : UINT;
	{attribute addProperty Name "Frm13Ctrl"}
	Frm13Ctrl AT %Q* : UINT;
	{attribute addProperty Name "Frm13WcCtrl"}
	Frm13WcCtrl AT %Q* : UINT;
	{attribute addProperty Name "Frm14Ctrl"}
	Frm14Ctrl AT %Q* : UINT;
	{attribute addProperty Name "Frm14WcCtrl"}
	Frm14WcCtrl AT %Q* : UINT;
	{attribute addProperty Name "Frm15Ctrl"}
	Frm15Ctrl AT %Q* : UINT;
	{attribute addProperty Name "Frm15WcCtrl"}
	Frm15WcCtrl AT %Q* : UINT;
	{attribute addProperty Name "Frm16Ctrl"}
	Frm16Ctrl AT %Q* : UINT;
	{attribute addProperty Name "Frm16WcCtrl"}
	Frm16WcCtrl AT %Q* : UINT;
	{attribute addProperty Name "Frm17Ctrl"}
	Frm17Ctrl AT %Q* : UINT;
	{attribute addProperty Name "Frm17WcCtrl"}
	Frm17WcCtrl AT %Q* : UINT;
	{attribute addProperty Name "Frm18Ctrl"}
	Frm18Ctrl AT %Q* : UINT;
	{attribute addProperty Name "Frm18WcCtrl"}
	Frm18WcCtrl AT %Q* : UINT;
	{attribute addProperty Name "Frm19Ctrl"}
	Frm19Ctrl AT %Q* : UINT;
	{attribute addProperty Name "Frm19WcCtrl"}
	Frm19WcCtrl AT %Q* : UINT;
	{attribute addProperty Name "Frm20Ctrl"}
	Frm20Ctrl AT %Q* : UINT;
	{attribute addProperty Name "Frm20WcCtrl"}
	Frm20WcCtrl AT %Q* : UINT;
	{attribute addProperty Name "Frm21Ctrl"}
	Frm21Ctrl AT %Q* : UINT;
	{attribute addProperty Name "Frm21WcCtrl"}
	Frm21WcCtrl AT %Q* : UINT;
	{attribute addProperty Name "Frm22Ctrl"}
	Frm22Ctrl AT %Q* : UINT;
	{attribute addProperty Name "Frm22WcCtrl"}
	Frm22WcCtrl AT %Q* : UINT;
	{attribute addProperty Name "Frm23Ctrl"}
	Frm23Ctrl AT %Q* : UINT;
	{attribute addProperty Name "Frm23WcCtrl"}
	Frm23WcCtrl AT %Q* : UINT;
	{attribute addProperty Name "Frm24Ctrl"}
	Frm24Ctrl AT %Q* : UINT;
	{attribute addProperty Name "Frm24WcCtrl"}
	Frm24WcCtrl AT %Q* : UINT;
	{attribute addProperty Name "Frm25Ctrl"}
	Frm25Ctrl AT %Q* : UINT;
	{attribute addProperty Name "Frm25WcCtrl"}
	Frm25WcCtrl AT %Q* : UINT;
END_STRUCT
END_TYPE

// ---- DUTs/IO/Boxes/EK1100_1FC0878B.TcDUT
{attribute 'GeneratedUsingTerminal: EK1100-0000-0018'}
{attribute addProperty BoxType "EK1100-0000-0018"}
{attribute addProperty Description "EK1100 EtherCAT Coupler (2A E-Bus)"}
{attribute addProperty Physics "YKY"}
{attribute addProperty Id "InfoDataAT %I*InfoData_6F19DB2B2"}
{attribute addProperty CRC "532711307"}
{attribute addProperty Size "2"}
TYPE EK1100_1FC0878B EXTENDS EtcSlaveBoxBase_77A0E4A7 :
STRUCT
	{attribute addProperty Name "InfoData"}
	InfoData : InfoData_6F19DB2B;
END_STRUCT
END_TYPE

// ---- DUTs/IO/Boxes/EK1122_1FC0878B.TcDUT
{attribute 'GeneratedUsingTerminal: EK1122-0000-0018'}
{attribute addProperty BoxType "EK1122-0000-0018"}
{attribute addProperty Description "EK1122 2 port EtherCAT junction"}
{attribute addProperty Physics "KYKY"}
{attribute addProperty Id "InfoDataAT %I*InfoData_6F19DB2B2"}
{attribute addProperty CRC "532711307"}
{attribute addProperty Size "2"}
TYPE EK1122_1FC0878B EXTENDS EtcSlaveTerminalBase_947E5A46 :
STRUCT
	{attribute addProperty Name "InfoData"}
	InfoData : InfoData_6F19DB2B;
END_STRUCT
END_TYPE

// ---- DUTs/IO/Boxes/EJ1100_1FC0878B.TcDUT
{attribute 'GeneratedUsingTerminal: EJ1100-0000-0018'}
{attribute addProperty BoxType "EJ1100-0000-0018"}
{attribute addProperty Description "EJ1100 EtherCAT Coupler (2.2A E-Bus)"}
{attribute addProperty Physics "YKY"}
{attribute addProperty Id "InfoDataAT %I*InfoData_6F19DB2B2"}
{attribute addProperty CRC "532711307"}
{attribute addProperty Size "2"}
TYPE EJ1100_1FC0878B EXTENDS EtcSlaveBoxBase_77A0E4A7 :
STRUCT
	{attribute addProperty Name "InfoData"}
	InfoData : InfoData_6F19DB2B;
END_STRUCT
END_TYPE

// ---- DUTs/IO/Boxes/EJ1101_D4DF6A22.TcDUT
{attribute 'GeneratedUsingTerminal: EJ1101-0022-0016'}
{attribute addProperty BoxType "EJ1101-0022-0016"}
{attribute addProperty Description "EJ1101-0022 EtherCAT Coupler (ID switch)"}
{attribute addProperty Physics "YKY"}
{attribute addProperty Id "WcStateAT %I*WcState_0B2B16F91InfoDataAT %I*InfoData_32EB74EA10"}
{attribute addProperty CRC "3571411490"}
{attribute addProperty Size "11"}
TYPE EJ1101_D4DF6A22 EXTENDS EtcSlaveBoxBase_77A0E4A7 :
STRUCT
	{attribute addProperty Name "WcState"}
	WcState : WcState_0B2B16F9;
	{attribute addProperty Name "InfoData"}
	InfoData : InfoData_32EB74EA;
END_STRUCT
END_TYPE

// ---- DUTs/IO/Boxes/EJ1008_78E8D3DD.TcDUT
{attribute 'GeneratedUsingTerminal: EJ1008-0000-0017'}
{attribute addProperty BoxType "EJ1008-0000-0017"}
{attribute addProperty Description "EJ1008 8Ch. Dig. Input 24V, 3ms"}
{attribute addProperty Physics "KK"}
{attribute addProperty Id "Channel_1AT %I*Channel_830843C11Channel_2AT %I*Channel_830843C11Channel_3AT %I*Channel_830843C11Channel_4AT %I*Channel_830843C11Channel_5AT %I*Channel_830843C11Channel_6AT %I*Channel_830843C11Channel_7AT %I*Channel_830843C11Channel_8AT %I*Channel_830843C11WcStateAT %I*WcState_9091E0EB2InfoDataAT %I*InfoData_6F19DB2B2"}
{attribute addProperty CRC "2028524509"}
{attribute addProperty Size "12"}
TYPE EJ1008_78E8D3DD EXTENDS EtcSlaveTerminalBase_947E5A46 :
STRUCT
	{attribute addProperty Name "Channel_1"}
	Channel_1 : Channel_830843C1;
	{attribute addProperty Name "Channel_2"}
	Channel_2 : Channel_830843C1;
	{attribute addProperty Name "Channel_3"}
	Channel_3 : Channel_830843C1;
	{attribute addProperty Name "Channel_4"}
	Channel_4 : Channel_830843C1;
	{attribute addProperty Name "Channel_5"}
	Channel_5 : Channel_830843C1;
	{attribute addProperty Name "Channel_6"}
	Channel_6 : Channel_830843C1;
	{attribute addProperty Name "Channel_7"}
	Channel_7 : Channel_830843C1;
	{attribute addProperty Name "Channel_8"}
	Channel_8 : Channel_830843C1;
	{attribute addProperty Name "WcState"}
	WcState : WcState_9091E0EB;
	{attribute addProperty Name "InfoData"}
	InfoData : InfoData_6F19DB2B;
END_STRUCT
END_TYPE

// ---- DUTs/IO/Boxes/EJ1128_78E8D3DD.TcDUT
{attribute 'GeneratedUsingTerminal: EJ1128-0000-0016'}
{attribute addProperty BoxType "EJ1128-0000-0016"}
{attribute addProperty Description "EJ1128 8Ch. Dig. Input 5V / 3.3V DC, 0.05µs"}
{attribute addProperty Physics "KK"}
{attribute addProperty Id "Channel_1AT %I*Channel_830843C11Channel_2AT %I*Channel_830843C11Channel_3AT %I*Channel_830843C11Channel_4AT %I*Channel_830843C11Channel_5AT %I*Channel_830843C11Channel_6AT %I*Channel_830843C11Channel_7AT %I*Channel_830843C11Channel_8AT %I*Channel_830843C11WcStateAT %I*WcState_9091E0EB2InfoDataAT %I*InfoData_6F19DB2B2"}
{attribute addProperty CRC "2028524509"}
{attribute addProperty Size "12"}
TYPE EJ1128_78E8D3DD EXTENDS EtcSlaveTerminalBase_947E5A46 :
STRUCT
	{attribute addProperty Name "Channel_1"}
	Channel_1 : Channel_830843C1;
	{attribute addProperty Name "Channel_2"}
	Channel_2 : Channel_830843C1;
	{attribute addProperty Name "Channel_3"}
	Channel_3 : Channel_830843C1;
	{attribute addProperty Name "Channel_4"}
	Channel_4 : Channel_830843C1;
	{attribute addProperty Name "Channel_5"}
	Channel_5 : Channel_830843C1;
	{attribute addProperty Name "Channel_6"}
	Channel_6 : Channel_830843C1;
	{attribute addProperty Name "Channel_7"}
	Channel_7 : Channel_830843C1;
	{attribute addProperty Name "Channel_8"}
	Channel_8 : Channel_830843C1;
	{attribute addProperty Name "WcState"}
	WcState : WcState_9091E0EB;
	{attribute addProperty Name "InfoData"}
	InfoData : InfoData_6F19DB2B;
END_STRUCT
END_TYPE

// ---- DUTs/IO/Boxes/EJ1809_32157CFD.TcDUT
{attribute 'GeneratedUsingTerminal: EJ1809-0000-0017'}
{attribute addProperty BoxType "EJ1809-0000-0017"}
{attribute addProperty Description "EJ1809 16Ch. Dig. Input 24V, 3ms"}
{attribute addProperty Physics "KK"}
{attribute addProperty Id "Channel_1AT %I*Channel_830843C11Channel_2AT %I*Channel_830843C11Channel_3AT %I*Channel_830843C11Channel_4AT %I*Channel_830843C11Channel_5AT %I*Channel_830843C11Channel_6AT %I*Channel_830843C11Channel_7AT %I*Channel_830843C11Channel_8AT %I*Channel_830843C11Channel_9AT %I*Channel_830843C11Channel_10AT %I*Channel_830843C11Channel_11AT %I*Channel_830843C11Channel_12AT %I*Channel_830843C11Channel_13AT %I*Channel_830843C11Channel_14AT %I*Channel_830843C11Channel_15AT %I*Channel_830843C11Channel_16AT %I*Channel_830843C11WcStateAT %I*WcState_9091E0EB2InfoDataAT %I*InfoData_6F19DB2B2"}
{attribute addProperty CRC "840269053"}
{attribute addProperty Size "20"}
TYPE EJ1809_32157CFD EXTENDS EtcSlaveTerminalBase_947E5A46 :
STRUCT
	{attribute addProperty Name "Channel_1"}
	Channel_1 : Channel_830843C1;
	{attribute addProperty Name "Channel_2"}
	Channel_2 : Channel_830843C1;
	{attribute addProperty Name "Channel_3"}
	Channel_3 : Channel_830843C1;
	{attribute addProperty Name "Channel_4"}
	Channel_4 : Channel_830843C1;
	{attribute addProperty Name "Channel_5"}
	Channel_5 : Channel_830843C1;
	{attribute addProperty Name "Channel_6"}
	Channel_6 : Channel_830843C1;
	{attribute addProperty Name "Channel_7"}
	Channel_7 : Channel_830843C1;
	{attribute addProperty Name "Channel_8"}
	Channel_8 : Channel_830843C1;
	{attribute addProperty Name "Channel_9"}
	Channel_9 : Channel_830843C1;
	{attribute addProperty Name "Channel_10"}
	Channel_10 : Channel_830843C1;
	{attribute addProperty Name "Channel_11"}
	Channel_11 : Channel_830843C1;
	{attribute addProperty Name "Channel_12"}
	Channel_12 : Channel_830843C1;
	{attribute addProperty Name "Channel_13"}
	Channel_13 : Channel_830843C1;
	{attribute addProperty Name "Channel_14"}
	Channel_14 : Channel_830843C1;
	{attribute addProperty Name "Channel_15"}
	Channel_15 : Channel_830843C1;
	{attribute addProperty Name "Channel_16"}
	Channel_16 : Channel_830843C1;
	{attribute addProperty Name "WcState"}
	WcState : WcState_9091E0EB;
	{attribute addProperty Name "InfoData"}
	InfoData : InfoData_6F19DB2B;
END_STRUCT
END_TYPE

// ---- DUTs/IO/Boxes/EJ1819_32157CFD.TcDUT
{attribute 'GeneratedUsingTerminal: EJ1819-0000-0017'}
{attribute addProperty BoxType "EJ1819-0000-0017"}
{attribute addProperty Description "EJ1819 16Ch. Dig. Input 24V, 10µs"}
{attribute addProperty Physics "KK"}
{attribute addProperty Id "Channel_1AT %I*Channel_830843C11Channel_2AT %I*Channel_830843C11Channel_3AT %I*Channel_830843C11Channel_4AT %I*Channel_830843C11Channel_5AT %I*Channel_830843C11Channel_6AT %I*Channel_830843C11Channel_7AT %I*Channel_830843C11Channel_8AT %I*Channel_830843C11Channel_9AT %I*Channel_830843C11Channel_10AT %I*Channel_830843C11Channel_11AT %I*Channel_830843C11Channel_12AT %I*Channel_830843C11Channel_13AT %I*Channel_830843C11Channel_14AT %I*Channel_830843C11Channel_15AT %I*Channel_830843C11Channel_16AT %I*Channel_830843C11WcStateAT %I*WcState_9091E0EB2InfoDataAT %I*InfoData_6F19DB2B2"}
{attribute addProperty CRC "840269053"}
{attribute addProperty Size "20"}
TYPE EJ1819_32157CFD EXTENDS EtcSlaveTerminalBase_947E5A46 :
STRUCT
	{attribute addProperty Name "Channel_1"}
	Channel_1 : Channel_830843C1;
	{attribute addProperty Name "Channel_2"}
	Channel_2 : Channel_830843C1;
	{attribute addProperty Name "Channel_3"}
	Channel_3 : Channel_830843C1;
	{attribute addProperty Name "Channel_4"}
	Channel_4 : Channel_830843C1;
	{attribute addProperty Name "Channel_5"}
	Channel_5 : Channel_830843C1;
	{attribute addProperty Name "Channel_6"}
	Channel_6 : Channel_830843C1;
	{attribute addProperty Name "Channel_7"}
	Channel_7 : Channel_830843C1;
	{attribute addProperty Name "Channel_8"}
	Channel_8 : Channel_830843C1;
	{attribute addProperty Name "Channel_9"}
	Channel_9 : Channel_830843C1;
	{attribute addProperty Name "Channel_10"}
	Channel_10 : Channel_830843C1;
	{attribute addProperty Name "Channel_11"}
	Channel_11 : Channel_830843C1;
	{attribute addProperty Name "Channel_12"}
	Channel_12 : Channel_830843C1;
	{attribute addProperty Name "Channel_13"}
	Channel_13 : Channel_830843C1;
	{attribute addProperty Name "Channel_14"}
	Channel_14 : Channel_830843C1;
	{attribute addProperty Name "Channel_15"}
	Channel_15 : Channel_830843C1;
	{attribute addProperty Name "Channel_16"}
	Channel_16 : Channel_830843C1;
	{attribute addProperty Name "WcState"}
	WcState : WcState_9091E0EB;
	{attribute addProperty Name "InfoData"}
	InfoData : InfoData_6F19DB2B;
END_STRUCT
END_TYPE

// ---- DUTs/IO/Boxes/EJ1859_7699BCF6.TcDUT
{attribute 'GeneratedUsingTerminal: EJ1859-0000-0017'}
{attribute addProperty BoxType "EJ1859-0000-0017"}
{attribute addProperty Description "EJ1859 8Ch. Dig. Input 24V, 3ms, 8Ch. Dig. Output 24V, 0.5A"}
{attribute addProperty Physics "KK"}
{attribute addProperty Id "Channel_1AT %I*Channel_830843C11Channel_2AT %I*Channel_830843C11Channel_3AT %I*Channel_830843C11Channel_4AT %I*Channel_830843C11Channel_5AT %I*Channel_830843C11Channel_6AT %I*Channel_830843C11Channel_7AT %I*Channel_830843C11Channel_8AT %I*Channel_830843C11Channel_9AT %Q*Channel_42CA91F71Channel_10AT %Q*Channel_42CA91F71Channel_11AT %Q*Channel_42CA91F71Channel_12AT %Q*Channel_42CA91F71Channel_13AT %Q*Channel_42CA91F71Channel_14AT %Q*Channel_42CA91F71Channel_15AT %Q*Channel_42CA91F71Channel_16AT %Q*Channel_42CA91F71WcStateAT %I*WcState_9091E0EB2InfoDataAT %I*InfoData_6F19DB2B2"}
{attribute addProperty CRC "1989786870"}
{attribute addProperty Size "20"}
TYPE EJ1859_7699BCF6 EXTENDS EtcSlaveTerminalBase_947E5A46 :
STRUCT
	{attribute addProperty Name "Channel_1"}
	Channel_1 : Channel_830843C1;
	{attribute addProperty Name "Channel_2"}
	Channel_2 : Channel_830843C1;
	{attribute addProperty Name "Channel_3"}
	Channel_3 : Channel_830843C1;
	{attribute addProperty Name "Channel_4"}
	Channel_4 : Channel_830843C1;
	{attribute addProperty Name "Channel_5"}
	Channel_5 : Channel_830843C1;
	{attribute addProperty Name "Channel_6"}
	Channel_6 : Channel_830843C1;
	{attribute addProperty Name "Channel_7"}
	Channel_7 : Channel_830843C1;
	{attribute addProperty Name "Channel_8"}
	Channel_8 : Channel_830843C1;
	{attribute addProperty Name "Channel_9"}
	Channel_9 : Channel_42CA91F7;
	{attribute addProperty Name "Channel_10"}
	Channel_10 : Channel_42CA91F7;
	{attribute addProperty Name "Channel_11"}
	Channel_11 : Channel_42CA91F7;
	{attribute addProperty Name "Channel_12"}
	Channel_12 : Channel_42CA91F7;
	{attribute addProperty Name "Channel_13"}
	Channel_13 : Channel_42CA91F7;
	{attribute addProperty Name "Channel_14"}
	Channel_14 : Channel_42CA91F7;
	{attribute addProperty Name "Channel_15"}
	Channel_15 : Channel_42CA91F7;
	{attribute addProperty Name "Channel_16"}
	Channel_16 : Channel_42CA91F7;
	{attribute addProperty Name "WcState"}
	WcState : WcState_9091E0EB;
	{attribute addProperty Name "InfoData"}
	InfoData : InfoData_6F19DB2B;
END_STRUCT
END_TYPE

